LIN {X 0,Y 247.88,Z 687.786,A -85,B 0,C 180,E1 -19070.205,E2 -19070.205} C_VEL
LIN {X 0,Y 249.229,Z 685.586,A -85,B 0,C 180,E1 -19073.523,E2 -19073.523} C_VEL
LIN {X 0,Y 251.079,Z 682.164,A -85,B 0,C 180,E1 -19076.79,E2 -19076.79} C_VEL
LIN {X 0,Y 253.652,Z 677.44,A -85,B 0,C 180,E1 -19080,E2 -19080} C_VEL
LIN {X 0,Y 256.854,Z 671.391,A -85,B 0,C 180,E1 -19083.137,E2 -19083.137} C_VEL
LIN {X 0,Y 260.765,Z 663.772,A -85,B 0,C 180,E1 -19086.188,E2 -19086.188} C_VEL
LIN {X 0,Y 264.838,Z 655.76,A -85,B 0,C 180,E1 -19088.777,E2 -19088.777} C_VEL
LIN {X 0,Y 267.711,Z 649.729,A -85,B 0,C 180,E1 -19090.41,E2 -19090.41} C_VEL
LIN {X 0,Y 268.928,Z 646.197,A -85,B 0,C 180,E1 -19091.383,E2 -19091.383} C_VEL
LIN {X 0,Y 270.336,Z 634.797,A -85,B 0,C 180,E1 -19094.806,E2 -19094.806} C_VEL
LIN {X 0,Y 271.75,Z 630.731,A -85,B 0,C 180,E1 -19095.669,E2 -19095.669} C_VEL
LIN {X 0,Y 276.734,Z 619.024,A -85,B 0,C 180,E1 -19097.552,E2 -19097.552} C_VEL
LIN {X 0,Y 281.807,Z 605.606,A -85,B 0,C 180,E1 -19099.296,E2 -19099.296} C_VEL
LIN {X 0,Y 286.56,Z 591.439,A -85,B 0,C 180,E1 -19100.778,E2 -19100.778} C_VEL
LIN {X 0,Y 290.862,Z 576.419,A -85,B 0,C 180,E1 -19101.994,E2 -19101.994} C_VEL
LIN {X 0,Y 294.362,Z 561.567,A -85,B 0,C 180,E1 -19102.921,E2 -19102.921} C_VEL
LIN {X 0,Y 297.341,Z 545.848,A -85,B 0,C 180,E1 -19103.645,E2 -19103.645} C_VEL
LIN {X 0,Y 308.948,Z 468.897,A -85,B 0,C 180,E1 -19106.327,E2 -19106.327} C_VEL
LIN {X 0,Y 307.213,Z 464.58,A -85,B 0,C 180,E1 -19107.92,E2 -19107.92} C_VEL
LIN {X 0,Y 305.635,Z 461.133,A -85,B 0,C 180,E1 -19109.693,E2 -19109.693} C_VEL
LIN {X 0,Y 304.433,Z 458.679,A -85,B 0,C 180,E1 -19111.555,E2 -19111.555} C_VEL
LIN {X 0,Y 303.585,Z 457.434,A -85,B 0,C 180,E1 -19113.752,E2 -19113.752} C_VEL
LIN {X 0,Y 303.382,Z 457.554,A -85,B 0,C 180,E1 -19115.824,E2 -19115.824} C_VEL
LIN {X 0,Y 303.96,Z 459.719,A -85,B 0,C 180,E1 -19118.511,E2 -19118.511} C_VEL
LIN {X 0,Y 304.573,Z 461.273,A -85,B 0,C 180,E1 -19119.738,E2 -19119.738} C_VEL
LIN {X 0,Y 305.975,Z 465.574,A -85,B 0,C 180,E1 -19121.819,E2 -19121.819} C_VEL
LIN {X 0,Y 307.607,Z 470.737,A -85,B 0,C 180,E1 -19123.621,E2 -19123.621} C_VEL
LIN {X 0,Y 308.482,Z 473.787,A -85,B 0,C 180,E1 -19124.465,E2 -19124.465} C_VEL
LIN {X 0,Y 296.017,Z 556.561,A -85,B 0,C 180,E1 -19127.358,E2 -19127.358} C_VEL
LIN {X 0,Y 292.723,Z 572.399,A -85,B 0,C 180,E1 -19128.104,E2 -19128.104} C_VEL
LIN {X 0,Y 288.495,Z 588.462,A -85,B 0,C 180,E1 -19129.101,E2 -19129.101} C_VEL
LIN {X 0,Y 283.818,Z 603.365,A -85,B 0,C 180,E1 -19130.328,E2 -19130.328} C_VEL
LIN {X 0,Y 278.241,Z 618.997,A -85,B 0,C 180,E1 -19131.996,E2 -19131.996} C_VEL
LIN {X 0,Y 272.662,Z 632.821,A -85,B 0,C 180,E1 -19133.868,E2 -19133.868} C_VEL
LIN {X 0,Y 266.356,Z 647.07,A -85,B 0,C 180,E1 -19136.349,E2 -19136.349} C_VEL
LIN {X 0,Y 261.075,Z 658.229,A -85,B 0,C 180,E1 -19138.786,E2 -19138.786} C_VEL
LIN {X 0,Y 255.836,Z 668.683,A -85,B 0,C 180,E1 -19141.623,E2 -19141.623} C_VEL
LIN {X 0,Y 251.787,Z 676.761,A -85,B 0,C 180,E1 -19144.362,E2 -19144.362} C_VEL
LIN {X 0,Y 248.026,Z 684.215,A -85,B 0,C 180,E1 -19147.507,E2 -19147.507} C_VEL
LIN {X 0,Y 244.834,Z 690.278,A -85,B 0,C 180,E1 -19150.722,E2 -19150.722} C_VEL
LIN {X 0,Y 242.981,Z 693.924,A -85,B 0,C 180,E1 -19153.185,E2 -19153.185} C_VEL
LIN {X 0,Y 241.338,Z 697.72,A -85,B 0,C 180,E1 -19156.526,E2 -19156.526} C_VEL
LIN {X 0,Y 240.312,Z 700.321,A -85,B 0,C 180,E1 -19159.891,E2 -19159.891} C_VEL
LIN {X 0,Y 239.794,Z 701.759,A -85,B 0,C 180,E1 -19163.265,E2 -19163.265} C_VEL
LIN {X 0,Y 239.757,Z 701.968,A -85,B 0,C 180,E1 -19166.637,E2 -19166.637} C_VEL
LIN {X 0,Y 239.893,Z 701.614,A -85,B 0,C 180,E1 -19168.319,E2 -19168.319} C_VEL
LIN {X 0,Y 239.926,Z 699.962,A -85,B 0,C 180,E1 -19171.676,E2 -19171.676} C_VEL
LIN {X 0,Y 239.941,Z 696.811,A -85,B 0,C 180,E1 -19175.209,E2 -19175.209} C_VEL
LIN {X 0,Y 240.087,Z 692.603,A -85,B 0,C 180,E1 -19178.414,E2 -19178.414} C_VEL
LIN {X 0,Y 240.543,Z 686.661,A -85,B 0,C 180,E1 -19181.799,E2 -19181.799} C_VEL
LIN {X 0,Y 241.434,Z 680.097,A -85,B 0,C 180,E1 -19184.753,E2 -19184.753} C_VEL
LIN {X 0,Y 242.744,Z 672.341,A -85,B 0,C 180,E1 -19187.608,E2 -19187.608} C_VEL
LIN {X 0,Y 244.273,Z 663.893,A -85,B 0,C 180,E1 -19190.194,E2 -19190.194} C_VEL
LIN {X 0,Y 246.574,Z 652.437,A -85,B 0,C 180,E1 -19193.071,E2 -19193.071} C_VEL
LIN {X 0,Y 248.822,Z 640.832,A -85,B 0,C 180,E1 -19195.466,E2 -19195.466} C_VEL
LIN {X 0,Y 251.171,Z 628.98,A -85,B 0,C 180,E1 -19197.493,E2 -19197.493} C_VEL
LIN {X 0,Y 253.722,Z 615.002,A -85,B 0,C 180,E1 -19199.447,E2 -19199.447} C_VEL
LIN {X 0,Y 256.022,Z 601.49,A -85,B 0,C 180,E1 -19200.974,E2 -19200.974} C_VEL
LIN {X 0,Y 258.145,Z 586.74,A -85,B 0,C 180,E1 -19202.304,E2 -19202.304} C_VEL
LIN {X 0,Y 260.031,Z 571.411,A -85,B 0,C 180,E1 -19203.353,E2 -19203.353} C_VEL
LIN {X 0,Y 261.5,Z 555.708,A -85,B 0,C 180,E1 -19204.124,E2 -19204.124} C_VEL
LIN {X 0,Y 268.174,Z 451.601,A -85,B 0,C 180,E1 -19207.78,E2 -19207.78} C_VEL
LIN {X 0,Y 267.38,Z 447.714,A -85,B 0,C 180,E1 -19208.028,E2 -19208.028} C_VEL
LIN {X 0,Y 257.514,Z 422.783,A -85,B 0,C 180,E1 -19210.24,E2 -19210.24} C_VEL
LIN {X 0,Y 249.94,Z 405.473,A -85,B 0,C 180,E1 -19212.023,E2 -19212.023} C_VEL
LIN {X 0,Y 243.579,Z 391.38,A -85,B 0,C 180,E1 -19213.612,E2 -19213.612} C_VEL
LIN {X 0,Y 241.939,Z 384.975,A -85,B 0,C 180,E1 -19216.029,E2 -19216.029} C_VEL
LIN {X 0,Y 241.93,Z 384.979,A -85,B 0,C 180,E1 -19220.276,E2 -19220.276} C_VEL
LIN {X 0,Y 241.966,Z 384.972,A -85,B 0,C 180,E1 -19224.486,E2 -19224.486} C_VEL
LIN {X 0,Y 241.936,Z 384.975,A -85,B 0,C 180,E1 -19228.475,E2 -19228.475} C_VEL
LIN {X 0,Y 241.938,Z 384.972,A -85,B 0,C 180,E1 -19232.305,E2 -19232.305} C_VEL
LIN {X 0,Y 241.969,Z 384.968,A -85,B 0,C 180,E1 -19236.007,E2 -19236.007} C_VEL
LIN {X 0,Y 241.971,Z 384.968,A -85,B 0,C 180,E1 -19239.603,E2 -19239.603} C_VEL
LIN {X 0,Y 242.092,Z 384.951,A -85,B 0,C 180,E1 -19243.324,E2 -19243.324} C_VEL
LIN {X 0,Y 242.139,Z 384.938,A -85,B 0,C 180,E1 -19248.278,E2 -19248.278} C_VEL
LIN {X 0,Y 242.354,Z 384.914,A -85,B 0,C 180,E1 -19251.663,E2 -19251.663} C_VEL
LIN {X 0,Y 242.382,Z 384.915,A -85,B 0,C 180,E1 -19253.34,E2 -19253.34} C_VEL
LIN {X 0,Y 242.603,Z 384.89,A -85,B 0,C 180,E1 -19258.34,E2 -19258.34} C_VEL
LIN {X 0,Y 242.603,Z 384.891,A -85,B 0,C 180,E1 -19261.661,E2 -19261.661} C_VEL
LIN {X 0,Y 242.386,Z 384.916,A -85,B 0,C 180,E1 -19266.661,E2 -19266.661} C_VEL
LIN {X 0,Y 242.247,Z 384.931,A -85,B 0,C 180,E1 -19270.025,E2 -19270.025} C_VEL
LIN {X 0,Y 242.095,Z 384.951,A -85,B 0,C 180,E1 -19275.146,E2 -19275.146} C_VEL
LIN {X 0,Y 242.007,Z 384.96,A -85,B 0,C 180,E1 -19278.63,E2 -19278.63} C_VEL
LIN {X 0,Y 241.961,Z 384.97,A -85,B 0,C 180,E1 -19282.185,E2 -19282.185} C_VEL
LIN {X 0,Y 241.975,Z 384.963,A -85,B 0,C 180,E1 -19285.828,E2 -19285.828} C_VEL
LIN {X 0,Y 241.952,Z 384.971,A -85,B 0,C 180,E1 -19289.591,E2 -19289.591} C_VEL
LIN {X 0,Y 241.969,Z 384.965,A -85,B 0,C 180,E1 -19293.495,E2 -19293.495} C_VEL
LIN {X 0,Y 241.97,Z 384.968,A -85,B 0,C 180,E1 -19297.586,E2 -19297.586} C_VEL
LIN {X 0,Y 241.91,Z 384.97,A -85,B 0,C 180,E1 -19301.929,E2 -19301.929} C_VEL
LIN {X 0,Y 241.892,Z 384.977,A -85,B 0,C 180,E1 -19306.583,E2 -19306.583} C_VEL
LIN {X 0,Y 241.968,Z 384.964,A -85,B 0,C 180,E1 -19311.649,E2 -19311.649} C_VEL
LIN {X 0,Y 241.968,Z 384.968,A -85,B 0,C 180,E1 -19314.489,E2 -19314.489} C_VEL
LIN {X 0,Y 241.943,Z 384.965,A -85,B 0,C 180,E1 -19318.479,E2 -19318.479} C_VEL
LIN {X 0,Y 241.948,Z 384.971,A -85,B 0,C 180,E1 -19322.308,E2 -19322.308} C_VEL
LIN {X 0,Y 241.984,Z 384.965,A -85,B 0,C 180,E1 -19326.011,E2 -19326.011} C_VEL
LIN {X 0,Y 242.019,Z 384.965,A -85,B 0,C 180,E1 -19329.609,E2 -19329.609} C_VEL
LIN {X 0,Y 242.115,Z 384.941,A -85,B 0,C 180,E1 -19333.319,E2 -19333.319} C_VEL
LIN {X 0,Y 242.155,Z 384.936,A -85,B 0,C 180,E1 -19336.577,E2 -19336.577} C_VEL
LIN {X 0,Y 242.343,Z 384.921,A -85,B 0,C 180,E1 -19340.407,E2 -19340.407} C_VEL
LIN {X 0,Y 242.398,Z 384.911,A -85,B 0,C 180,E1 -19343.343,E2 -19343.343} C_VEL
LIN {X 0,Y 242.622,Z 384.888,A -85,B 0,C 180,E1 -19348.343,E2 -19348.343} C_VEL
LIN {X 0,Y 242.621,Z 384.883,A -85,B 0,C 180,E1 -19351.662,E2 -19351.662} C_VEL
LIN {X 0,Y 242.403,Z 384.916,A -85,B 0,C 180,E1 -19356.662,E2 -19356.662} C_VEL
LIN {X 0,Y 242.27,Z 384.93,A -85,B 0,C 180,E1 -19360.026,E2 -19360.026} C_VEL
LIN {X 0,Y 242.112,Z 384.948,A -85,B 0,C 180,E1 -19365.147,E2 -19365.147} C_VEL
LIN {X 0,Y 242.044,Z 384.956,A -85,B 0,C 180,E1 -19368.629,E2 -19368.629} C_VEL
LIN {X 0,Y 242.007,Z 384.962,A -85,B 0,C 180,E1 -19372.183,E2 -19372.183} C_VEL
LIN {X 0,Y 241.995,Z 384.966,A -85,B 0,C 180,E1 -19376.756,E2 -19376.756} C_VEL
LIN {X 0,Y 242.034,Z 384.961,A -85,B 0,C 180,E1 -19377.628,E2 -19377.628} C_VEL
LIN {X 0,Y 243.106,Z 387.957,A -85,B 0,C 180,E1 -19377.964,E2 -19377.964} C_VEL
LIN {X 0,Y 254.638,Z 409.921,A -85,B 0,C 180,E1 -19380.548,E2 -19380.548} C_VEL
LIN {X 0,Y 260.374,Z 422.165,A -85,B 0,C 180,E1 -19381.812,E2 -19381.812} C_VEL
LIN {X 0,Y 268.163,Z 441.082,A -85,B 0,C 180,E1 -19383.506,E2 -19383.506} C_VEL
LIN {X 0,Y 261.391,Z 544.984,A -85,B 0,C 180,E1 -19387.16,E2 -19387.16} C_VEL
LIN {X 0,Y 259.827,Z 560.878,A -85,B 0,C 180,E1 -19388.019,E2 -19388.019} C_VEL
LIN {X 0,Y 257.976,Z 576.825,A -85,B 0,C 180,E1 -19389.221,E2 -19389.221} C_VEL
LIN {X 0,Y 255.654,Z 592.523,A -85,B 0,C 180,E1 -19390.758,E2 -19390.758} C_VEL
LIN {X 0,Y 253.408,Z 605.906,A -85,B 0,C 180,E1 -19392.403,E2 -19392.403} C_VEL
LIN {X 0,Y 250.916,Z 619.48,A -85,B 0,C 180,E1 -19394.448,E2 -19394.448} C_VEL
LIN {X 0,Y 248.588,Z 631.789,A -85,B 0,C 180,E1 -19396.717,E2 -19396.717} C_VEL
LIN {X 0,Y 246.446,Z 642.171,A -85,B 0,C 180,E1 -19399.011,E2 -19399.011} C_VEL
LIN {X 0,Y 244.425,Z 652.702,A -85,B 0,C 180,E1 -19401.815,E2 -19401.815} C_VEL
LIN {X 0,Y 242.777,Z 661.39,A -85,B 0,C 180,E1 -19404.621,E2 -19404.621} C_VEL
LIN {X 0,Y 241.533,Z 668.857,A -85,B 0,C 180,E1 -19407.55,E2 -19407.55} C_VEL
LIN {X 0,Y 240.741,Z 674.529,A -85,B 0,C 180,E1 -19410.245,E2 -19410.245} C_VEL
LIN {X 0,Y 240.186,Z 679.262,A -85,B 0,C 180,E1 -19413.028,E2 -19413.028} C_VEL
LIN {X 0,Y 239.715,Z 682.915,A -85,B 0,C 180,E1 -19415.766,E2 -19415.766} C_VEL
LIN {X 0,Y 239.447,Z 686.389,A -85,B 0,C 180,E1 -19419.377,E2 -19419.377} C_VEL
LIN {X 0,Y 239.498,Z 688.397,A -85,B 0,C 180,E1 -19422.935,E2 -19422.935} C_VEL
LIN {X 0,Y 239.883,Z 689.056,A -85,B 0,C 180,E1 -19426.444,E2 -19426.444} C_VEL
LIN {X 0,Y 240.675,Z 688.451,A -85,B 0,C 180,E1 -19429.909,E2 -19429.909} C_VEL
LIN {X 0,Y 242.053,Z 686.612,A -85,B 0,C 180,E1 -19433.33,E2 -19433.33} C_VEL
LIN {X 0,Y 243.902,Z 683.528,A -85,B 0,C 180,E1 -19436.696,E2 -19436.696} C_VEL
LIN {X 0,Y 246.518,Z 679.203,A -85,B 0,C 180,E1 -19440,E2 -19440} C_VEL
LIN {X 0,Y 249.783,Z 673.54,A -85,B 0,C 180,E1 -19443.225,E2 -19443.225} C_VEL
LIN {X 0,Y 253.794,Z 666.466,A -85,B 0,C 180,E1 -19446.359,E2 -19446.359} C_VEL
LIN {X 0,Y 257.915,Z 658.897,A -85,B 0,C 180,E1 -19449.014,E2 -19449.014} C_VEL
LIN {X 0,Y 262.61,Z 649.918,A -85,B 0,C 180,E1 -19451.578,E2 -19451.578} C_VEL
LIN {X 0,Y 267.686,Z 639.572,A -85,B 0,C 180,E1 -19453.972,E2 -19453.972} C_VEL
LIN {X 0,Y 271.75,Z 630.731,A -85,B 0,C 180,E1 -19455.669,E2 -19455.669} C_VEL
LIN {X 0,Y 273.213,Z 626.626,A -85,B 0,C 180,E1 -19456.512,E2 -19456.512} C_VEL
LIN {X 0,Y 275.152,Z 614.753,A -85,B 0,C 180,E1 -19459.27,E2 -19459.27} C_VEL
LIN {X 0,Y 276.382,Z 610.304,A -85,B 0,C 180,E1 -19460.027,E2 -19460.027} C_VEL
LIN {X 0,Y 276.968,Z 608.722,A -85,B 0,C 180,E1 -19460.234,E2 -19460.234} C_VEL
LIN {X 0,Y 282.024,Z 594.812,A -85,B 0,C 180,E1 -19461.744,E2 -19461.744} C_VEL
LIN {X 0,Y 286.38,Z 581.125,A -85,B 0,C 180,E1 -19462.928,E2 -19462.928} C_VEL
LIN {X 0,Y 290.018,Z 567.604,A -85,B 0,C 180,E1 -19463.852,E2 -19463.852} C_VEL
LIN {X 0,Y 293.521,Z 551.339,A -85,B 0,C 180,E1 -19464.692,E2 -19464.692} C_VEL
LIN {X 0,Y 306.022,Z 473.195,A -85,B 0,C 180,E1 -19467.45,E2 -19467.45} C_VEL
LIN {X 0,Y 304.117,Z 468.309,A -85,B 0,C 180,E1 -19469.655,E2 -19469.655} C_VEL
LIN {X 0,Y 302.839,Z 465.531,A -85,B 0,C 180,E1 -19471.741,E2 -19471.741} C_VEL
LIN {X 0,Y 302.066,Z 464.347,A -85,B 0,C 180,E1 -19473.945,E2 -19473.945} C_VEL
LIN {X 0,Y 301.907,Z 464.592,A -85,B 0,C 180,E1 -19475.977,E2 -19475.977} C_VEL
LIN {X 0,Y 302.48,Z 466.851,A -85,B 0,C 180,E1 -19478.591,E2 -19478.591} C_VEL
LIN {X 0,Y 302.861,Z 468.094,A -85,B 0,C 180,E1 -19479.481,E2 -19479.481} C_VEL
LIN {X 0,Y 303.977,Z 471.983,A -85,B 0,C 180,E1 -19481.373,E2 -19481.373} C_VEL
LIN {X 0,Y 305.294,Z 476.638,A -85,B 0,C 180,E1 -19483.026,E2 -19483.026} C_VEL
LIN {X 0,Y 305.571,Z 477.721,A -85,B 0,C 180,E1 -19483.342,E2 -19483.342} C_VEL
LIN {X 0,Y 293.012,Z 556.809,A -85,B 0,C 180,E1 -19486.104,E2 -19486.104} C_VEL
LIN {X 0,Y 289.914,Z 571.167,A -85,B 0,C 180,E1 -19486.776,E2 -19486.776} C_VEL
LIN {X 0,Y 285.639,Z 586.713,A -85,B 0,C 180,E1 -19487.716,E2 -19487.716} C_VEL
LIN {X 0,Y 280.729,Z 601.757,A -85,B 0,C 180,E1 -19488.914,E2 -19488.914} C_VEL
LIN {X 0,Y 275.464,Z 615.934,A -85,B 0,C 180,E1 -19490.367,E2 -19490.367} C_VEL
LIN {X 0,Y 269.538,Z 630.011,A -85,B 0,C 180,E1 -19492.21,E2 -19492.21} C_VEL
LIN {X 0,Y 264.115,Z 641.993,A -85,B 0,C 180,E1 -19494.166,E2 -19494.166} C_VEL
LIN {X 0,Y 259.08,Z 652.225,A -85,B 0,C 180,E1 -19496.211,E2 -19496.211} C_VEL
LIN {X 0,Y 253.7,Z 662.524,A -85,B 0,C 180,E1 -19498.705,E2 -19498.705} C_VEL
LIN {X 0,Y 248.935,Z 671.26,A -85,B 0,C 180,E1 -19501.316,E2 -19501.316} C_VEL
LIN {X 0,Y 244.378,Z 679.622,A -85,B 0,C 180,E1 -19504.442,E2 -19504.442} C_VEL
LIN {X 0,Y 240.604,Z 686.476,A -85,B 0,C 180,E1 -19507.681,E2 -19507.681} C_VEL
LIN {X 0,Y 237.393,Z 692.002,A -85,B 0,C 180,E1 -19510.992,E2 -19510.992} C_VEL
LIN {X 0,Y 235.258,Z 696.205,A -85,B 0,C 180,E1 -19514.401,E2 -19514.401} C_VEL
LIN {X 0,Y 233.715,Z 699.218,A -85,B 0,C 180,E1 -19517.846,E2 -19517.846} C_VEL
LIN {X 0,Y 232.949,Z 701.078,A -85,B 0,C 180,E1 -19521.321,E2 -19521.321} C_VEL
LIN {X 0,Y 232.646,Z 701.784,A -85,B 0,C 180,E1 -19524.798,E2 -19524.798} C_VEL
LIN {X 0,Y 232.798,Z 701.286,A -85,B 0,C 180,E1 -19528.267,E2 -19528.267} C_VEL
LIN {X 0,Y 232.848,Z 700.548,A -85,B 0,C 180,E1 -19529.997,E2 -19529.997} C_VEL
LIN {X 0,Y 232.858,Z 699.488,A -85,B 0,C 180,E1 -19531.727,E2 -19531.727} C_VEL
LIN {X 0,Y 232.878,Z 696.368,A -85,B 0,C 180,E1 -19535.192,E2 -19535.192} C_VEL
LIN {X 0,Y 233.02,Z 691.824,A -85,B 0,C 180,E1 -19538.671,E2 -19538.671} C_VEL
LIN {X 0,Y 233.545,Z 685.73,A -85,B 0,C 180,E1 -19542.158,E2 -19542.158} C_VEL
LIN {X 0,Y 234.483,Z 678.999,A -85,B 0,C 180,E1 -19545.201,E2 -19545.201} C_VEL
LIN {X 0,Y 235.945,Z 670.799,A -85,B 0,C 180,E1 -19548.223,E2 -19548.223} C_VEL
LIN {X 0,Y 237.867,Z 660.853,A -85,B 0,C 180,E1 -19551.216,E2 -19551.216} C_VEL
LIN {X 0,Y 239.931,Z 650.663,A -85,B 0,C 180,E1 -19553.748,E2 -19553.748} C_VEL
LIN {X 0,Y 242.137,Z 639.638,A -85,B 0,C 180,E1 -19556.037,E2 -19556.037} C_VEL
LIN {X 0,Y 244.514,Z 627.848,A -85,B 0,C 180,E1 -19558.074,E2 -19558.074} C_VEL
LIN {X 0,Y 246.881,Z 615.258,A -85,B 0,C 180,E1 -19559.876,E2 -19559.876} C_VEL
LIN {X 0,Y 249.229,Z 601.848,A -85,B 0,C 180,E1 -19561.442,E2 -19561.442} C_VEL
LIN {X 0,Y 251.34,Z 587.946,A -85,B 0,C 180,E1 -19562.746,E2 -19562.746} C_VEL
LIN {X 0,Y 253.369,Z 572.224,A -85,B 0,C 180,E1 -19563.87,E2 -19563.87} C_VEL
LIN {X 0,Y 254.826,Z 556.973,A -85,B 0,C 180,E1 -19564.665,E2 -19564.665} C_VEL
LIN {X 0,Y 261.743,Z 452.264,A -85,B 0,C 180,E1 -19568.45,E2 -19568.45} C_VEL
LIN {X 0,Y 259.763,Z 446.226,A -85,B 0,C 180,E1 -19568.937,E2 -19568.937} C_VEL
LIN {X 0,Y 249.571,Z 420.785,A -85,B 0,C 180,E1 -19571.354,E2 -19571.354} C_VEL
LIN {X 0,Y 239.424,Z 398.251,A -85,B 0,C 180,E1 -19573.825,E2 -19573.825} C_VEL
LIN {X 0,Y 236.247,Z 391.245,A -85,B 0,C 180,E1 -19574.684,E2 -19574.684} C_VEL
LIN {X 0,Y 234.906,Z 385.85,A -85,B 0,C 180,E1 -19576.78,E2 -19576.78} C_VEL
LIN {X 0,Y 234.907,Z 385.851,A -85,B 0,C 180,E1 -19581.077,E2 -19581.077} C_VEL
LIN {X 0,Y 234.913,Z 385.849,A -85,B 0,C 180,E1 -19585.36,E2 -19585.36} C_VEL
LIN {X 0,Y 234.882,Z 385.852,A -85,B 0,C 180,E1 -19589.426,E2 -19589.426} C_VEL
LIN {X 0,Y 234.927,Z 385.841,A -85,B 0,C 180,E1 -19593.82,E2 -19593.82} C_VEL
LIN {X 0,Y 234.923,Z 385.845,A -85,B 0,C 180,E1 -19598.962,E2 -19598.962} C_VEL
LIN {X 0,Y 235.036,Z 385.829,A -85,B 0,C 180,E1 -19603.097,E2 -19603.097} C_VEL
LIN {X 0,Y 235.071,Z 385.821,A -85,B 0,C 180,E1 -19607.92,E2 -19607.92} C_VEL
LIN {X 0,Y 235.291,Z 385.793,A -85,B 0,C 180,E1 -19611.411,E2 -19611.411} C_VEL
LIN {X 0,Y 235.333,Z 385.793,A -85,B 0,C 180,E1 -19613.14,E2 -19613.14} C_VEL
LIN {X 0,Y 235.562,Z 385.767,A -85,B 0,C 180,E1 -19618.291,E2 -19618.291} C_VEL
LIN {X 0,Y 235.562,Z 385.768,A -85,B 0,C 180,E1 -19621.71,E2 -19621.71} C_VEL
LIN {X 0,Y 235.338,Z 385.794,A -85,B 0,C 180,E1 -19626.861,E2 -19626.861} C_VEL
LIN {X 0,Y 235.171,Z 385.811,A -85,B 0,C 180,E1 -19630.33,E2 -19630.33} C_VEL
LIN {X 0,Y 235.047,Z 385.831,A -85,B 0,C 180,E1 -19635.611,E2 -19635.611} C_VEL
LIN {X 0,Y 234.948,Z 385.839,A -85,B 0,C 180,E1 -19639.211,E2 -19639.211} C_VEL
LIN {X 0,Y 234.905,Z 385.846,A -85,B 0,C 180,E1 -19642.889,E2 -19642.889} C_VEL
LIN {X 0,Y 234.911,Z 385.842,A -85,B 0,C 180,E1 -19646.665,E2 -19646.665} C_VEL
LIN {X 0,Y 234.884,Z 385.85,A -85,B 0,C 180,E1 -19650.575,E2 -19650.575} C_VEL
LIN {X 0,Y 234.915,Z 385.84,A -85,B 0,C 180,E1 -19654.641,E2 -19654.641} C_VEL
LIN {X 0,Y 234.903,Z 385.847,A -85,B 0,C 180,E1 -19658.937,E2 -19658.937} C_VEL
LIN {X 0,Y 234.853,Z 385.848,A -85,B 0,C 180,E1 -19663.495,E2 -19663.495} C_VEL
LIN {X 0,Y 234.845,Z 385.855,A -85,B 0,C 180,E1 -19666.508,E2 -19666.508} C_VEL
LIN {X 0,Y 234.912,Z 385.839,A -85,B 0,C 180,E1 -19671.081,E2 -19671.081} C_VEL
LIN {X 0,Y 234.917,Z 385.847,A -85,B 0,C 180,E1 -19675.363,E2 -19675.363} C_VEL
LIN {X 0,Y 234.89,Z 385.845,A -85,B 0,C 180,E1 -19679.43,E2 -19679.43} C_VEL
LIN {X 0,Y 234.937,Z 385.844,A -85,B 0,C 180,E1 -19683.824,E2 -19683.824} C_VEL
LIN {X 0,Y 234.966,Z 385.841,A -85,B 0,C 180,E1 -19688.969,E2 -19688.969} C_VEL
LIN {X 0,Y 235.056,Z 385.822,A -85,B 0,C 180,E1 -19693.095,E2 -19693.095} C_VEL
LIN {X 0,Y 235.111,Z 385.82,A -85,B 0,C 180,E1 -19697.925,E2 -19697.925} C_VEL
LIN {X 0,Y 235.313,Z 385.799,A -85,B 0,C 180,E1 -19701.414,E2 -19701.414} C_VEL
LIN {X 0,Y 235.349,Z 385.79,A -85,B 0,C 180,E1 -19703.142,E2 -19703.142} C_VEL
LIN {X 0,Y 235.581,Z 385.765,A -85,B 0,C 180,E1 -19708.293,E2 -19708.293} C_VEL
LIN {X 0,Y 235.58,Z 385.759,A -85,B 0,C 180,E1 -19711.712,E2 -19711.712} C_VEL
LIN {X 0,Y 235.354,Z 385.795,A -85,B 0,C 180,E1 -19716.863,E2 -19716.863} C_VEL
LIN {X 0,Y 235.216,Z 385.809,A -85,B 0,C 180,E1 -19720.33,E2 -19720.33} C_VEL
LIN {X 0,Y 235.064,Z 385.829,A -85,B 0,C 180,E1 -19725.612,E2 -19725.612} C_VEL
LIN {X 0,Y 234.987,Z 385.836,A -85,B 0,C 180,E1 -19729.21,E2 -19729.21} C_VEL
LIN {X 0,Y 234.946,Z 385.843,A -85,B 0,C 180,E1 -19732.887,E2 -19732.887} C_VEL
LIN {X 0,Y 234.947,Z 385.844,A -85,B 0,C 180,E1 -19736.622,E2 -19736.622} C_VEL
LIN {X 0,Y 236.012,Z 388.749,A -85,B 0,C 180,E1 -19736.951,E2 -19736.951} C_VEL
LIN {X 0,Y 245.134,Z 405.869,A -85,B 0,C 180,E1 -19739.113,E2 -19739.113} C_VEL
LIN {X 0,Y 254.074,Z 424.079,A -85,B 0,C 180,E1 -19741.121,E2 -19741.121} C_VEL
LIN {X 0,Y 261.689,Z 442.792,A -85,B 0,C 180,E1 -19742.858,E2 -19742.858} C_VEL
LIN {X 0,Y 254.839,Z 545.121,A -85,B 0,C 180,E1 -19746.561,E2 -19746.561} C_VEL
LIN {X 0,Y 253.405,Z 559.639,A -85,B 0,C 180,E1 -19747.348,E2 -19747.348} C_VEL
LIN {X 0,Y 251.53,Z 575.326,A -85,B 0,C 180,E1 -19748.523,E2 -19748.523} C_VEL
LIN {X 0,Y 249.326,Z 590.237,A -85,B 0,C 180,E1 -19749.971,E2 -19749.971} C_VEL
LIN {X 0,Y 246.957,Z 604.162,A -85,B 0,C 180,E1 -19751.665,E2 -19751.665} C_VEL
LIN {X 0,Y 244.422,Z 617.892,A -85,B 0,C 180,E1 -19753.732,E2 -19753.732} C_VEL
LIN {X 0,Y 241.913,Z 630.767,A -85,B 0,C 180,E1 -19756.11,E2 -19756.11} C_VEL
LIN {X 0,Y 239.506,Z 642.24,A -85,B 0,C 180,E1 -19758.682,E2 -19758.682} C_VEL
LIN {X 0,Y 237.407,Z 652.772,A -85,B 0,C 180,E1 -19761.561,E2 -19761.561} C_VEL
LIN {X 0,Y 235.738,Z 661.481,A -85,B 0,C 180,E1 -19764.454,E2 -19764.454} C_VEL
LIN {X 0,Y 234.342,Z 669.777,A -85,B 0,C 180,E1 -19767.836,E2 -19767.836} C_VEL
LIN {X 0,Y 233.419,Z 676.327,A -85,B 0,C 180,E1 -19771.2,E2 -19771.2} C_VEL
LIN {X 0,Y 232.888,Z 680.716,A -85,B 0,C 180,E1 -19774.051,E2 -19774.051} C_VEL
LIN {X 0,Y 232.454,Z 684.107,A -85,B 0,C 180,E1 -19776.856,E2 -19776.856} C_VEL
LIN {X 0,Y 232.326,Z 687.238,A -85,B 0,C 180,E1 -19780.563,E2 -19780.563} C_VEL
LIN {X 0,Y 232.501,Z 688.912,A -85,B 0,C 180,E1 -19784.213,E2 -19784.213} C_VEL
LIN {X 0,Y 233.018,Z 689.267,A -85,B 0,C 180,E1 -19787.811,E2 -19787.811} C_VEL
LIN {X 0,Y 234.303,Z 688.173,A -85,B 0,C 180,E1 -19791.841,E2 -19791.841} C_VEL
LIN {X 0,Y 235.672,Z 686.289,A -85,B 0,C 180,E1 -19794.867,E2 -19794.867} C_VEL
LIN {X 0,Y 237.956,Z 682.995,A -85,B 0,C 180,E1 -19798.307,E2 -19798.307} C_VEL
LIN {X 0,Y 240.926,Z 678.434,A -85,B 0,C 180,E1 -19801.671,E2 -19801.671} C_VEL
LIN {X 0,Y 244.642,Z 672.569,A -85,B 0,C 180,E1 -19804.944,E2 -19804.944} C_VEL
LIN {X 0,Y 249.142,Z 665.161,A -85,B 0,C 180,E1 -19808.108,E2 -19808.108} C_VEL
LIN {X 0,Y 253.725,Z 657.352,A -85,B 0,C 180,E1 -19810.776,E2 -19810.776} C_VEL
LIN {X 0,Y 258.818,Z 648.03,A -85,B 0,C 180,E1 -19813.344,E2 -19813.344} C_VEL
LIN {X 0,Y 264.514,Z 637.022,A -85,B 0,C 180,E1 -19815.803,E2 -19815.803} C_VEL
LIN {X 0,Y 270.253,Z 624.759,A -85,B 0,C 180,E1 -19817.987,E2 -19817.987} C_VEL
LIN {X 0,Y 275.602,Z 612.271,A -85,B 0,C 180,E1 -19819.786,E2 -19819.786} C_VEL
LIN {X 0,Y 276.968,Z 608.722,A -85,B 0,C 180,E1 -19820.234,E2 -19820.234} C_VEL
LIN {X 0,Y 277.872,Z 605.639,A -85,B 0,C 180,E1 -19820.725,E2 -19820.725} C_VEL
LIN {X 0,Y 278.565,Z 596.621,A -85,B 0,C 180,E1 -19822.794,E2 -19822.794} C_VEL
LIN {X 0,Y 279.424,Z 593.394,A -85,B 0,C 180,E1 -19823.237,E2 -19823.237} C_VEL
LIN {X 0,Y 284.267,Z 578.423,A -85,B 0,C 180,E1 -19824.463,E2 -19824.463} C_VEL
LIN {X 0,Y 288.074,Z 564.569,A -85,B 0,C 180,E1 -19825.353,E2 -19825.353} C_VEL
LIN {X 0,Y 291.605,Z 548.16,A -85,B 0,C 180,E1 -19826.133,E2 -19826.133} C_VEL
LIN {X 0,Y 303.352,Z 478.07,A -85,B 0,C 180,E1 -19828.57,E2 -19828.57} C_VEL
LIN {X 0,Y 302.289,Z 474.84,A -85,B 0,C 180,E1 -19830.055,E2 -19830.055} C_VEL
LIN {X 0,Y 301.249,Z 472.363,A -85,B 0,C 180,E1 -19831.928,E2 -19831.928} C_VEL
LIN {X 0,Y 300.682,Z 471.449,A -85,B 0,C 180,E1 -19833.356,E2 -19833.356} C_VEL
LIN {X 0,Y 300.404,Z 471.447,A -85,B 0,C 180,E1 -19835.794,E2 -19835.794} C_VEL
LIN {X 0,Y 300.889,Z 473.712,A -85,B 0,C 180,E1 -19838.407,E2 -19838.407} C_VEL
LIN {X 0,Y 301.298,Z 475.468,A -85,B 0,C 180,E1 -19839.516,E2 -19839.516} C_VEL
LIN {X 0,Y 302.161,Z 478.839,A -85,B 0,C 180,E1 -19841.105,E2 -19841.105} C_VEL
LIN {X 0,Y 302.933,Z 481.857,A -85,B 0,C 180,E1 -19842.18,E2 -19842.18} C_VEL
LIN {X 0,Y 290.514,Z 556.084,A -85,B 0,C 180,E1 -19844.773,E2 -19844.773} C_VEL
LIN {X 0,Y 287.297,Z 570.283,A -85,B 0,C 180,E1 -19845.429,E2 -19845.429} C_VEL
LIN {X 0,Y 283.012,Z 585.339,A -85,B 0,C 180,E1 -19846.315,E2 -19846.315} C_VEL
LIN {X 0,Y 277.871,Z 600.527,A -85,B 0,C 180,E1 -19847.48,E2 -19847.48} C_VEL
LIN {X 0,Y 272.49,Z 614.341,A -85,B 0,C 180,E1 -19848.874,E2 -19848.874} C_VEL
LIN {X 0,Y 266.239,Z 628.608,A -85,B 0,C 180,E1 -19850.686,E2 -19850.686} C_VEL
LIN {X 0,Y 261.391,Z 638.78,A -85,B 0,C 180,E1 -19852.287,E2 -19852.287} C_VEL
LIN {X 0,Y 255.076,Z 650.971,A -85,B 0,C 180,E1 -19854.645,E2 -19854.645} C_VEL
LIN {X 0,Y 249.316,Z 661.336,A -85,B 0,C 180,E1 -19857.134,E2 -19857.134} C_VEL
LIN {X 0,Y 243.775,Z 670.822,A -85,B 0,C 180,E1 -19859.976,E2 -19859.976} C_VEL
LIN {X 0,Y 239.161,Z 678.628,A -85,B 0,C 180,E1 -19862.901,E2 -19862.901} C_VEL
LIN {X 0,Y 235.007,Z 685.573,A -85,B 0,C 180,E1 -19866.186,E2 -19866.186} C_VEL
LIN {X 0,Y 231.458,Z 691.171,A -85,B 0,C 180,E1 -19869.56,E2 -19869.56} C_VEL
LIN {X 0,Y 229.35,Z 694.553,A -85,B 0,C 180,E1 -19872.153,E2 -19872.153} C_VEL
LIN {X 0,Y 227.494,Z 698.022,A -85,B 0,C 180,E1 -19875.689,E2 -19875.689} C_VEL
LIN {X 0,Y 226.228,Z 700.271,A -85,B 0,C 180,E1 -19879.255,E2 -19879.255} C_VEL
LIN {X 0,Y 225.652,Z 701.393,A -85,B 0,C 180,E1 -19882.841,E2 -19882.841} C_VEL
LIN {X 0,Y 225.59,Z 701.356,A -85,B 0,C 180,E1 -19886.425,E2 -19886.425} C_VEL
LIN {X 0,Y 225.706,Z 700.893,A -85,B 0,C 180,E1 -19888.213,E2 -19888.213} C_VEL
LIN {X 0,Y 225.781,Z 700.119,A -85,B 0,C 180,E1 -19889.997,E2 -19889.997} C_VEL
LIN {X 0,Y 225.791,Z 699.008,A -85,B 0,C 180,E1 -19891.781,E2 -19891.781} C_VEL
LIN {X 0,Y 225.795,Z 695.735,A -85,B 0,C 180,E1 -19895.355,E2 -19895.355} C_VEL
LIN {X 0,Y 225.951,Z 691.018,A -85,B 0,C 180,E1 -19898.944,E2 -19898.944} C_VEL
LIN {X 0,Y 226.548,Z 684.741,A -85,B 0,C 180,E1 -19902.539,E2 -19902.539} C_VEL
LIN {X 0,Y 227.554,Z 677.81,A -85,B 0,C 180,E1 -19905.676,E2 -19905.676} C_VEL
LIN {X 0,Y 229.124,Z 669.405,A -85,B 0,C 180,E1 -19908.785,E2 -19908.785} C_VEL
LIN {X 0,Y 231.132,Z 659.229,A -85,B 0,C 180,E1 -19911.866,E2 -19911.866} C_VEL
LIN {X 0,Y 233.294,Z 648.781,A -85,B 0,C 180,E1 -19914.467,E2 -19914.467} C_VEL
LIN {X 0,Y 235.698,Z 637.487,A -85,B 0,C 180,E1 -19916.804,E2 -19916.804} C_VEL
LIN {X 0,Y 238.43,Z 624.031,A -85,B 0,C 180,E1 -19919.098,E2 -19919.098} C_VEL
LIN {X 0,Y 240.935,Z 610.748,A -85,B 0,C 180,E1 -19920.935,E2 -19920.935} C_VEL
LIN {X 0,Y 243.587,Z 595.469,A -85,B 0,C 180,E1 -19922.624,E2 -19922.624} C_VEL
LIN {X 0,Y 245.798,Z 579.823,A -85,B 0,C 180,E1 -19923.954,E2 -19923.954} C_VEL
LIN {X 0,Y 247.654,Z 563.903,A -85,B 0,C 180,E1 -19924.948,E2 -19924.948} C_VEL
LIN {X 0,Y 249.069,Z 546.189,A -85,B 0,C 180,E1 -19925.711,E2 -19925.711} C_VEL
LIN {X 0,Y 255.379,Z 453.331,A -85,B 0,C 180,E1 -19929.134,E2 -19929.134} C_VEL
LIN {X 0,Y 246.046,Z 429.434,A -85,B 0,C 180,E1 -19931.394,E2 -19931.394} C_VEL
LIN {X 0,Y 236.311,Z 406.954,A -85,B 0,C 180,E1 -19933.839,E2 -19933.839} C_VEL
LIN {X 0,Y 228.915,Z 390.974,A -85,B 0,C 180,E1 -19935.851,E2 -19935.851} C_VEL
LIN {X 0,Y 227.816,Z 386.734,A -85,B 0,C 180,E1 -19937.583,E2 -19937.583} C_VEL
LIN {X 0,Y 227.828,Z 386.735,A -85,B 0,C 180,E1 -19941.906,E2 -19941.906} C_VEL
LIN {X 0,Y 227.867,Z 386.729,A -85,B 0,C 180,E1 -19946.376,E2 -19946.376} C_VEL
LIN {X 0,Y 227.859,Z 386.727,A -85,B 0,C 180,E1 -19950.43,E2 -19950.43} C_VEL
LIN {X 0,Y 227.858,Z 386.72,A -85,B 0,C 180,E1 -19954.418,E2 -19954.418} C_VEL
LIN {X 0,Y 227.906,Z 386.722,A -85,B 0,C 180,E1 -19958.282,E2 -19958.282} C_VEL
LIN {X 0,Y 227.996,Z 386.709,A -85,B 0,C 180,E1 -19963.894,E2 -19963.894} C_VEL
LIN {X 0,Y 228.112,Z 386.681,A -85,B 0,C 180,E1 -19969.348,E2 -19969.348} C_VEL
LIN {X 0,Y 228.285,Z 386.671,A -85,B 0,C 180,E1 -19972.927,E2 -19972.927} C_VEL
LIN {X 0,Y 228.52,Z 386.644,A -85,B 0,C 180,E1 -19978.238,E2 -19978.238} C_VEL
LIN {X 0,Y 228.52,Z 386.645,A -85,B 0,C 180,E1 -19981.763,E2 -19981.763} C_VEL
LIN {X 0,Y 228.291,Z 386.672,A -85,B 0,C 180,E1 -19987.074,E2 -19987.074} C_VEL
LIN {X 0,Y 228.112,Z 386.69,A -85,B 0,C 180,E1 -19990.653,E2 -19990.653} C_VEL
LIN {X 0,Y 227.997,Z 386.706,A -85,B 0,C 180,E1 -19996.107,E2 -19996.107} C_VEL
LIN {X 0,Y 227.908,Z 386.722,A -85,B 0,C 180,E1 -20001.719,E2 -20001.719} C_VEL
LIN {X 0,Y 227.89,Z 386.717,A -85,B 0,C 180,E1 -20006.583,E2 -20006.583} C_VEL
LIN {X 0,Y 227.859,Z 386.726,A -85,B 0,C 180,E1 -20010.281,E2 -20010.281} C_VEL
LIN {X 0,Y 227.867,Z 386.719,A -85,B 0,C 180,E1 -20013.723,E2 -20013.723} C_VEL
LIN {X 0,Y 227.831,Z 386.73,A -85,B 0,C 180,E1 -20018.094,E2 -20018.094} C_VEL
LIN {X 0,Y 227.784,Z 386.726,A -85,B 0,C 180,E1 -20022.749,E2 -20022.749} C_VEL
LIN {X 0,Y 227.776,Z 386.736,A -85,B 0,C 180,E1 -20027.254,E2 -20027.254} C_VEL
LIN {X 0,Y 227.831,Z 386.726,A -85,B 0,C 180,E1 -20031.91,E2 -20031.91} C_VEL
LIN {X 0,Y 227.873,Z 386.722,A -85,B 0,C 180,E1 -20036.381,E2 -20036.381} C_VEL
LIN {X 0,Y 227.867,Z 386.724,A -85,B 0,C 180,E1 -20040.434,E2 -20040.434} C_VEL
LIN {X 0,Y 227.869,Z 386.721,A -85,B 0,C 180,E1 -20044.422,E2 -20044.422} C_VEL
LIN {X 0,Y 227.94,Z 386.717,A -85,B 0,C 180,E1 -20048.288,E2 -20048.288} C_VEL
LIN {X 0,Y 228.024,Z 386.687,A -85,B 0,C 180,E1 -20053.898,E2 -20053.898} C_VEL
LIN {X 0,Y 228.068,Z 386.693,A -85,B 0,C 180,E1 -20057.546,E2 -20057.546} C_VEL
LIN {X 0,Y 228.254,Z 386.677,A -85,B 0,C 180,E1 -20061.147,E2 -20061.147} C_VEL
LIN {X 0,Y 228.302,Z 386.667,A -85,B 0,C 180,E1 -20062.93,E2 -20062.93} C_VEL
LIN {X 0,Y 228.539,Z 386.643,A -85,B 0,C 180,E1 -20068.24,E2 -20068.24} C_VEL
LIN {X 0,Y 228.538,Z 386.636,A -85,B 0,C 180,E1 -20071.765,E2 -20071.765} C_VEL
LIN {X 0,Y 228.307,Z 386.673,A -85,B 0,C 180,E1 -20077.075,E2 -20077.075} C_VEL
LIN {X 0,Y 228.145,Z 386.689,A -85,B 0,C 180,E1 -20080.654,E2 -20080.654} C_VEL
LIN {X 0,Y 228.015,Z 386.708,A -85,B 0,C 180,E1 -20086.108,E2 -20086.108} C_VEL
LIN {X 0,Y 227.956,Z 386.712,A -85,B 0,C 180,E1 -20091.716,E2 -20091.716} C_VEL
LIN {X 0,Y 227.887,Z 386.721,A -85,B 0,C 180,E1 -20095.582,E2 -20095.582} C_VEL
LIN {X 0,Y 228.967,Z 389.691,A -85,B 0,C 180,E1 -20095.919,E2 -20095.919} C_VEL
LIN {X 0,Y 236.787,Z 404.157,A -85,B 0,C 180,E1 -20097.849,E2 -20097.849} C_VEL
LIN {X 0,Y 247.403,Z 425.27,A -85,B 0,C 180,E1 -20100.333,E2 -20100.333} C_VEL
LIN {X 0,Y 255.318,Z 444.708,A -85,B 0,C 180,E1 -20102.202,E2 -20102.202} C_VEL
LIN {X 0,Y 248.307,Z 545.265,A -85,B 0,C 180,E1 -20105.93,E2 -20105.93} C_VEL
LIN {X 0,Y 246.656,Z 561.176,A -85,B 0,C 180,E1 -20106.838,E2 -20106.838} C_VEL
LIN {X 0,Y 244.802,Z 576.313,A -85,B 0,C 180,E1 -20108.028,E2 -20108.028} C_VEL
LIN {X 0,Y 242.58,Z 590.75,A -85,B 0,C 180,E1 -20109.479,E2 -20109.479} C_VEL
LIN {X 0,Y 239.969,Z 605.635,A -85,B 0,C 180,E1 -20111.367,E2 -20111.367} C_VEL
LIN {X 0,Y 237.328,Z 619.128,A -85,B 0,C 180,E1 -20113.487,E2 -20113.487} C_VEL
LIN {X 0,Y 234.827,Z 631.721,A -85,B 0,C 180,E1 -20115.916,E2 -20115.916} C_VEL
LIN {X 0,Y 232.352,Z 643.214,A -85,B 0,C 180,E1 -20118.603,E2 -20118.603} C_VEL
LIN {X 0,Y 230.418,Z 652.74,A -85,B 0,C 180,E1 -20121.297,E2 -20121.297} C_VEL
LIN {X 0,Y 228.677,Z 661.491,A -85,B 0,C 180,E1 -20124.272,E2 -20124.272} C_VEL
LIN {X 0,Y 227.384,Z 668.957,A -85,B 0,C 180,E1 -20127.352,E2 -20127.352} C_VEL
LIN {X 0,Y 226.517,Z 674.875,A -85,B 0,C 180,E1 -20130.317,E2 -20130.317} C_VEL
LIN {X 0,Y 225.963,Z 679.509,A -85,B 0,C 180,E1 -20133.192,E2 -20133.192} C_VEL
LIN {X 0,Y 225.465,Z 683.22,A -85,B 0,C 180,E1 -20136.094,E2 -20136.094} C_VEL
LIN {X 0,Y 225.267,Z 686.742,A -85,B 0,C 180,E1 -20139.928,E2 -20139.928} C_VEL
LIN {X 0,Y 225.348,Z 688.808,A -85,B 0,C 180,E1 -20143.698,E2 -20143.698} C_VEL
LIN {X 0,Y 225.858,Z 689.553,A -85,B 0,C 180,E1 -20147.419,E2 -20147.419} C_VEL
LIN {X 0,Y 226.884,Z 689.044,A -85,B 0,C 180,E1 -20151.09,E2 -20151.09} C_VEL
LIN {X 0,Y 228.465,Z 687.305,A -85,B 0,C 180,E1 -20154.704,E2 -20154.704} C_VEL
LIN {X 0,Y 230.753,Z 684.351,A -85,B 0,C 180,E1 -20158.254,E2 -20158.254} C_VEL
LIN {X 0,Y 233.788,Z 680.208,A -85,B 0,C 180,E1 -20161.722,E2 -20161.722} C_VEL
LIN {X 0,Y 237.569,Z 674.745,A -85,B 0,C 180,E1 -20165.091,E2 -20165.091} C_VEL
LIN {X 0,Y 242.155,Z 667.904,A -85,B 0,C 180,E1 -20168.343,E2 -20168.343} C_VEL
LIN {X 0,Y 246.86,Z 660.573,A -85,B 0,C 180,E1 -20171.079,E2 -20171.079} C_VEL
LIN {X 0,Y 252.082,Z 651.932,A -85,B 0,C 180,E1 -20173.708,E2 -20173.708} C_VEL
LIN {X 0,Y 257.933,Z 641.573,A -85,B 0,C 180,E1 -20176.217,E2 -20176.217} C_VEL
LIN {X 0,Y 264.294,Z 629.262,A -85,B 0,C 180,E1 -20178.608,E2 -20178.608} C_VEL
LIN {X 0,Y 269.857,Z 617.35,A -85,B 0,C 180,E1 -20180.46,E2 -20180.46} C_VEL
LIN {X 0,Y 275.642,Z 603.53,A -85,B 0,C 180,E1 -20182.191,E2 -20182.191} C_VEL
LIN {X 0,Y 279.424,Z 593.394,A -85,B 0,C 180,E1 -20183.237,E2 -20183.237} C_VEL
LIN {X 0,Y 280.913,Z 588.416,A -85,B 0,C 180,E1 -20183.815,E2 -20183.815} C_VEL
LIN {X 0,Y 283.61,Z 573.276,A -85,B 0,C 180,E1 -20186.01,E2 -20186.01} C_VEL
LIN {X 0,Y 284.985,Z 567.147,A -85,B 0,C 180,E1 -20186.559,E2 -20186.559} C_VEL
LIN {X 0,Y 288.913,Z 550.598,A -85,B 0,C 180,E1 -20187.381,E2 -20187.381} C_VEL
LIN {X 0,Y 300.89,Z 482.824,A -85,B 0,C 180,E1 -20189.734,E2 -20189.734} C_VEL
LIN {X 0,Y 300.23,Z 480.93,A -85,B 0,C 180,E1 -20190.828,E2 -20190.828} C_VEL
LIN {X 0,Y 299.504,Z 478.973,A -85,B 0,C 180,E1 -20192.477,E2 -20192.477} C_VEL
LIN {X 0,Y 299.007,Z 478.22,A -85,B 0,C 180,E1 -20194.34,E2 -20194.34} C_VEL
LIN {X 0,Y 298.899,Z 478.623,A -85,B 0,C 180,E1 -20196.002,E2 -20196.002} C_VEL
LIN {X 0,Y 299.396,Z 480.83,A -85,B 0,C 180,E1 -20198.471,E2 -20198.471} C_VEL
LIN {X 0,Y 300.182,Z 484.699,A -85,B 0,C 180,E1 -20200.421,E2 -20200.421} C_VEL
LIN {X 0,Y 300.466,Z 486.129,A -85,B 0,C 180,E1 -20200.996,E2 -20200.996} C_VEL
LIN {X 0,Y 288.367,Z 555.09,A -85,B 0,C 180,E1 -20203.397,E2 -20203.397} C_VEL
LIN {X 0,Y 284.741,Z 570.433,A -85,B 0,C 180,E1 -20204.094,E2 -20204.094} C_VEL
LIN {X 0,Y 280.285,Z 585.415,A -85,B 0,C 180,E1 -20204.966,E2 -20204.966} C_VEL
LIN {X 0,Y 274.952,Z 600.295,A -85,B 0,C 180,E1 -20206.103,E2 -20206.103} C_VEL
LIN {X 0,Y 268.628,Z 615.623,A -85,B 0,C 180,E1 -20207.645,E2 -20207.645} C_VEL
LIN {X 0,Y 262.647,Z 628.437,A -85,B 0,C 180,E1 -20209.287,E2 -20209.287} C_VEL
LIN {X 0,Y 256.071,Z 641.252,A -85,B 0,C 180,E1 -20211.36,E2 -20211.36} C_VEL
LIN {X 0,Y 249.523,Z 652.955,A -85,B 0,C 180,E1 -20213.735,E2 -20213.735} C_VEL
LIN {X 0,Y 242.731,Z 664.229,A -85,B 0,C 180,E1 -20216.622,E2 -20216.622} C_VEL
LIN {X 0,Y 236.745,Z 673.595,A -85,B 0,C 180,E1 -20219.689,E2 -20219.689} C_VEL
LIN {X 0,Y 231.749,Z 681.36,A -85,B 0,C 180,E1 -20222.94,E2 -20222.94} C_VEL
LIN {X 0,Y 227.535,Z 687.685,A -85,B 0,C 180,E1 -20226.323,E2 -20226.323} C_VEL
LIN {X 0,Y 223.993,Z 692.772,A -85,B 0,C 180,E1 -20229.807,E2 -20229.807} C_VEL
LIN {X 0,Y 221.476,Z 696.629,A -85,B 0,C 180,E1 -20233.403,E2 -20233.403} C_VEL
LIN {X 0,Y 219.749,Z 699.348,A -85,B 0,C 180,E1 -20237.061,E2 -20237.061} C_VEL
LIN {X 0,Y 218.837,Z 700.881,A -85,B 0,C 180,E1 -20240.757,E2 -20240.757} C_VEL
LIN {X 0,Y 218.479,Z 701.26,A -85,B 0,C 180,E1 -20244.459,E2 -20244.459} C_VEL
LIN {X 0,Y 218.617,Z 700.469,A -85,B 0,C 180,E1 -20248.155,E2 -20248.155} C_VEL
LIN {X 0,Y 218.716,Z 699.614,A -85,B 0,C 180,E1 -20249.997,E2 -20249.997} C_VEL
LIN {X 0,Y 218.726,Z 698.431,A -85,B 0,C 180,E1 -20251.839,E2 -20251.839} C_VEL
LIN {X 0,Y 218.727,Z 695.041,A -85,B 0,C 180,E1 -20255.529,E2 -20255.529} C_VEL
LIN {X 0,Y 218.908,Z 690.184,A -85,B 0,C 180,E1 -20259.234,E2 -20259.234} C_VEL
LIN {X 0,Y 219.559,Z 683.701,A -85,B 0,C 180,E1 -20262.945,E2 -20262.945} C_VEL
LIN {X 0,Y 220.651,Z 676.61,A -85,B 0,C 180,E1 -20266.179,E2 -20266.179} C_VEL
LIN {X 0,Y 222.268,Z 667.974,A -85,B 0,C 180,E1 -20269.387,E2 -20269.387} C_VEL
LIN {X 0,Y 224.472,Z 657.521,A -85,B 0,C 180,E1 -20272.55,E2 -20272.55} C_VEL
LIN {X 0,Y 226.703,Z 646.784,A -85,B 0,C 180,E1 -20275.227,E2 -20275.227} C_VEL
LIN {X 0,Y 229.296,Z 635.194,A -85,B 0,C 180,E1 -20277.615,E2 -20277.615} C_VEL
LIN {X 0,Y 231.853,Z 622.636,A -85,B 0,C 180,E1 -20279.756,E2 -20279.756} C_VEL
LIN {X 0,Y 234.447,Z 609.105,A -85,B 0,C 180,E1 -20281.638,E2 -20281.638} C_VEL
LIN {X 0,Y 237.02,Z 594.43,A -85,B 0,C 180,E1 -20283.264,E2 -20283.264} C_VEL
LIN {X 0,Y 239.207,Z 579.513,A -85,B 0,C 180,E1 -20284.558,E2 -20284.558} C_VEL
LIN {X 0,Y 241.138,Z 563.178,A -85,B 0,C 180,E1 -20285.604,E2 -20285.604} C_VEL
LIN {X 0,Y 242.628,Z 544.57,A -85,B 0,C 180,E1 -20286.424,E2 -20286.424} C_VEL
LIN {X 0,Y 249.032,Z 455.148,A -85,B 0,C 180,E1 -20289.824,E2 -20289.824} C_VEL
LIN {X 0,Y 239.71,Z 431.398,A -85,B 0,C 180,E1 -20292.13,E2 -20292.13} C_VEL
LIN {X 0,Y 230.857,Z 410.788,A -85,B 0,C 180,E1 -20294.456,E2 -20294.456} C_VEL
LIN {X 0,Y 221.629,Z 390.787,A -85,B 0,C 180,E1 -20297.047,E2 -20297.047} C_VEL
LIN {X 0,Y 220.734,Z 387.617,A -85,B 0,C 180,E1 -20298.405,E2 -20298.405} C_VEL
LIN {X 0,Y 220.814,Z 387.607,A -85,B 0,C 180,E1 -20302.791,E2 -20302.791} C_VEL
LIN {X 0,Y 220.799,Z 387.607,A -85,B 0,C 180,E1 -20307.242,E2 -20307.242} C_VEL
LIN {X 0,Y 220.783,Z 387.608,A -85,B 0,C 180,E1 -20311.479,E2 -20311.479} C_VEL
LIN {X 0,Y 220.79,Z 387.602,A -85,B 0,C 180,E1 -20315.556,E2 -20315.556} C_VEL
LIN {X 0,Y 220.834,Z 387.6,A -85,B 0,C 180,E1 -20319.509,E2 -20319.509} C_VEL
LIN {X 0,Y 220.957,Z 387.583,A -85,B 0,C 180,E1 -20323.366,E2 -20323.366} C_VEL
LIN {X 0,Y 221.037,Z 387.562,A -85,B 0,C 180,E1 -20329.003,E2 -20329.003} C_VEL
LIN {X 0,Y 221.222,Z 387.551,A -85,B 0,C 180,E1 -20332.7,E2 -20332.7} C_VEL
LIN {X 0,Y 221.454,Z 387.523,A -85,B 0,C 180,E1 -20338.182,E2 -20338.182} C_VEL
LIN {X 0,Y 221.454,Z 387.524,A -85,B 0,C 180,E1 -20341.819,E2 -20341.819} C_VEL
LIN {X 0,Y 221.228,Z 387.552,A -85,B 0,C 180,E1 -20347.301,E2 -20347.301} C_VEL
LIN {X 0,Y 221.037,Z 387.57,A -85,B 0,C 180,E1 -20350.998,E2 -20350.998} C_VEL
LIN {X 0,Y 220.958,Z 387.579,A -85,B 0,C 180,E1 -20356.635,E2 -20356.635} C_VEL
LIN {X 0,Y 220.835,Z 387.601,A -85,B 0,C 180,E1 -20360.492,E2 -20360.492} C_VEL
LIN {X 0,Y 220.792,Z 387.6,A -85,B 0,C 180,E1 -20364.445,E2 -20364.445} C_VEL
LIN {X 0,Y 220.785,Z 387.606,A -85,B 0,C 180,E1 -20368.522,E2 -20368.522} C_VEL
LIN {X 0,Y 220.801,Z 387.599,A -85,B 0,C 180,E1 -20372.759,E2 -20372.759} C_VEL
LIN {X 0,Y 220.791,Z 387.604,A -85,B 0,C 180,E1 -20377.277,E2 -20377.277} C_VEL
LIN {X 0,Y 220.746,Z 387.605,A -85,B 0,C 180,E1 -20381.959,E2 -20381.959} C_VEL
LIN {X 0,Y 220.746,Z 387.611,A -85,B 0,C 180,E1 -20385.543,E2 -20385.543} C_VEL
LIN {X 0,Y 220.774,Z 387.6,A -85,B 0,C 180,E1 -20390.46,E2 -20390.46} C_VEL
LIN {X 0,Y 220.819,Z 387.6,A -85,B 0,C 180,E1 -20392.796,E2 -20392.796} C_VEL
LIN {X 0,Y 220.806,Z 387.602,A -85,B 0,C 180,E1 -20397.246,E2 -20397.246} C_VEL
LIN {X 0,Y 220.792,Z 387.607,A -85,B 0,C 180,E1 -20401.484,E2 -20401.484} C_VEL
LIN {X 0,Y 220.804,Z 387.601,A -85,B 0,C 180,E1 -20405.561,E2 -20405.561} C_VEL
LIN {X 0,Y 220.869,Z 387.599,A -85,B 0,C 180,E1 -20409.515,E2 -20409.515} C_VEL
LIN {X 0,Y 220.979,Z 387.569,A -85,B 0,C 180,E1 -20413.37,E2 -20413.37} C_VEL
LIN {X 0,Y 221.005,Z 387.57,A -85,B 0,C 180,E1 -20417.141,E2 -20417.141} C_VEL
LIN {X 0,Y 221.195,Z 387.556,A -85,B 0,C 180,E1 -20420.862,E2 -20420.862} C_VEL
LIN {X 0,Y 221.112,Z 387.552,A -85,B 0,C 180,E1 -20424.531,E2 -20424.531} C_VEL
LIN {X 0,Y 221.472,Z 387.524,A -85,B 0,C 180,E1 -20428.184,E2 -20428.184} C_VEL
LIN {X 0,Y 221.472,Z 387.515,A -85,B 0,C 180,E1 -20431.821,E2 -20431.821} C_VEL
LIN {X 0,Y 221.244,Z 387.553,A -85,B 0,C 180,E1 -20437.303,E2 -20437.303} C_VEL
LIN {X 0,Y 221.065,Z 387.572,A -85,B 0,C 180,E1 -20440.999,E2 -20440.999} C_VEL
LIN {X 0,Y 220.976,Z 387.584,A -85,B 0,C 180,E1 -20446.636,E2 -20446.636} C_VEL
LIN {X 0,Y 220.881,Z 387.597,A -85,B 0,C 180,E1 -20450.49,E2 -20450.49} C_VEL
LIN {X 0,Y 220.839,Z 387.6,A -85,B 0,C 180,E1 -20454.441,E2 -20454.441} C_VEL
LIN {X 0,Y 221.866,Z 390.532,A -85,B 0,C 180,E1 -20454.819,E2 -20454.819} C_VEL
LIN {X 0,Y 224.793,Z 395.709,A -85,B 0,C 180,E1 -20455.587,E2 -20455.587} C_VEL
LIN {X 0,Y 234.687,Z 414.558,A -85,B 0,C 180,E1 -20458.072,E2 -20458.072} C_VEL
LIN {X 0,Y 242.778,Z 431.254,A -85,B 0,C 180,E1 -20460.021,E2 -20460.021} C_VEL
LIN {X 0,Y 248.894,Z 446.32,A -85,B 0,C 180,E1 -20461.496,E2 -20461.496} C_VEL
LIN {X 0,Y 241.746,Z 545.121,A -85,B 0,C 180,E1 -20465.285,E2 -20465.285} C_VEL
LIN {X 0,Y 240.088,Z 561.029,A -85,B 0,C 180,E1 -20466.212,E2 -20466.212} C_VEL
LIN {X 0,Y 238.126,Z 576.465,A -85,B 0,C 180,E1 -20467.451,E2 -20467.451} C_VEL
LIN {X 0,Y 235.821,Z 591.062,A -85,B 0,C 180,E1 -20468.958,E2 -20468.958} C_VEL
LIN {X 0,Y 233.257,Z 605.267,A -85,B 0,C 180,E1 -20470.798,E2 -20470.798} C_VEL
LIN {X 0,Y 230.548,Z 618.874,A -85,B 0,C 180,E1 -20472.977,E2 -20472.977} C_VEL
LIN {X 0,Y 227.905,Z 631.78,A -85,B 0,C 180,E1 -20475.522,E2 -20475.522} C_VEL
LIN {X 0,Y 225.401,Z 643.162,A -85,B 0,C 180,E1 -20478.249,E2 -20478.249} C_VEL
LIN {X 0,Y 223.432,Z 652.712,A -85,B 0,C 180,E1 -20481.016,E2 -20481.016} C_VEL
LIN {X 0,Y 221.627,Z 661.51,A -85,B 0,C 180,E1 -20484.079,E2 -20484.079} C_VEL
LIN {X 0,Y 220.165,Z 669.909,A -85,B 0,C 180,E1 -20487.677,E2 -20487.677} C_VEL
LIN {X 0,Y 219.222,Z 676.514,A -85,B 0,C 180,E1 -20491.256,E2 -20491.256} C_VEL
LIN {X 0,Y 218.67,Z 680.786,A -85,B 0,C 180,E1 -20494.151,E2 -20494.151} C_VEL
LIN {X 0,Y 218.234,Z 684.362,A -85,B 0,C 180,E1 -20497.266,E2 -20497.266} C_VEL
LIN {X 0,Y 218.155,Z 686.148,A -85,B 0,C 180,E1 -20499.244,E2 -20499.244} C_VEL
LIN {X 0,Y 218.194,Z 688.604,A -85,B 0,C 180,E1 -20503.148,E2 -20503.148} C_VEL
LIN {X 0,Y 218.679,Z 689.699,A -85,B 0,C 180,E1 -20506.998,E2 -20506.998} C_VEL
LIN {X 0,Y 219.648,Z 689.541,A -85,B 0,C 180,E1 -20510.794,E2 -20510.794} C_VEL
LIN {X 0,Y 221.258,Z 688.184,A -85,B 0,C 180,E1 -20514.531,E2 -20514.531} C_VEL
LIN {X 0,Y 223.574,Z 685.668,A -85,B 0,C 180,E1 -20518.198,E2 -20518.198} C_VEL
LIN {X 0,Y 226.647,Z 681.923,A -85,B 0,C 180,E1 -20521.776,E2 -20521.776} C_VEL
LIN {X 0,Y 230.505,Z 676.91,A -85,B 0,C 180,E1 -20525.248,E2 -20525.248} C_VEL
LIN {X 0,Y 235.191,Z 670.532,A -85,B 0,C 180,E1 -20528.592,E2 -20528.592} C_VEL
LIN {X 0,Y 240.751,Z 662.635,A -85,B 0,C 180,E1 -20531.791,E2 -20531.791} C_VEL
LIN {X 0,Y 246.178,Z 654.311,A -85,B 0,C 180,E1 -20534.465,E2 -20534.465} C_VEL
LIN {X 0,Y 252.267,Z 644.438,A -85,B 0,C 180,E1 -20537.009,E2 -20537.009} C_VEL
LIN {X 0,Y 257.911,Z 634.474,A -85,B 0,C 180,E1 -20539.086,E2 -20539.086} C_VEL
LIN {X 0,Y 264.024,Z 622.632,A -85,B 0,C 180,E1 -20541.111,E2 -20541.111} C_VEL
LIN {X 0,Y 270.285,Z 609.098,A -85,B 0,C 180,E1 -20542.956,E2 -20542.956} C_VEL
LIN {X 0,Y 276.497,Z 593.762,A -85,B 0,C 180,E1 -20544.596,E2 -20544.596} C_VEL
LIN {X 0,Y 281.937,Z 577.798,A -85,B 0,C 180,E1 -20545.885,E2 -20545.885} C_VEL
LIN {X 0,Y 284.985,Z 567.147,A -85,B 0,C 180,E1 -20546.559,E2 -20546.559} C_VEL
LIN {X 0,Y 285.738,Z 563.585,A -85,B 0,C 180,E1 -20546.899,E2 -20546.899} C_VEL
LIN {X 0,Y 286.735,Z 552.878,A -85,B 0,C 180,E1 -20548.54,E2 -20548.54} C_VEL
LIN {X 0,Y 287.311,Z 549.195,A -85,B 0,C 180,E1 -20548.807,E2 -20548.807} C_VEL
LIN {X 0,Y 298.596,Z 488.224,A -85,B 0,C 180,E1 -20550.887,E2 -20550.887} C_VEL
LIN {X 0,Y 298.641,Z 487.861,A -85,B 0,C 180,E1 -20550.924,E2 -20550.924} C_VEL
LIN {X 0,Y 297.923,Z 485.821,A -85,B 0,C 180,E1 -20552.671,E2 -20552.671} C_VEL
LIN {X 0,Y 297.534,Z 485.166,A -85,B 0,C 180,E1 -20554.233,E2 -20554.233} C_VEL
LIN {X 0,Y 297.392,Z 485.516,A -85,B 0,C 180,E1 -20555.851,E2 -20555.851} C_VEL
LIN {X 0,Y 297.726,Z 487.449,A -85,B 0,C 180,E1 -20558.062,E2 -20558.062} C_VEL
LIN {X 0,Y 298.261,Z 490.775,A -85,B 0,C 180,E1 -20559.809,E2 -20559.809} C_VEL
LIN {X 0,Y 286.279,Z 555.616,A -85,B 0,C 180,E1 -20562.047,E2 -20562.047} C_VEL
LIN {X 0,Y 282.657,Z 570.141,A -85,B 0,C 180,E1 -20562.687,E2 -20562.687} C_VEL
LIN {X 0,Y 277.782,Z 585.661,A -85,B 0,C 180,E1 -20563.593,E2 -20563.593} C_VEL
LIN {X 0,Y 272.697,Z 599.258,A -85,B 0,C 180,E1 -20564.603,E2 -20564.603} C_VEL
LIN {X 0,Y 266.665,Z 613.359,A -85,B 0,C 180,E1 -20565.961,E2 -20565.961} C_VEL
LIN {X 0,Y 260.377,Z 626.285,A -85,B 0,C 180,E1 -20567.56,E2 -20567.56} C_VEL
LIN {X 0,Y 253.867,Z 638.467,A -85,B 0,C 180,E1 -20569.413,E2 -20569.413} C_VEL
LIN {X 0,Y 246.868,Z 650.392,A -85,B 0,C 180,E1 -20571.74,E2 -20571.74} C_VEL
LIN {X 0,Y 240.467,Z 660.634,A -85,B 0,C 180,E1 -20574.228,E2 -20574.228} C_VEL
LIN {X 0,Y 235.412,Z 668.141,A -85,B 0,C 180,E1 -20576.472,E2 -20576.472} C_VEL
LIN {X 0,Y 230.732,Z 674.802,A -85,B 0,C 180,E1 -20578.812,E2 -20578.812} C_VEL
LIN {X 0,Y 225.502,Z 682.24,A -85,B 0,C 180,E1 -20582.126,E2 -20582.126} C_VEL
LIN {X 0,Y 221.063,Z 688.373,A -85,B 0,C 180,E1 -20585.585,E2 -20585.585} C_VEL
LIN {X 0,Y 217.331,Z 693.189,A -85,B 0,C 180,E1 -20589.16,E2 -20589.16} C_VEL
LIN {X 0,Y 214.618,Z 696.841,A -85,B 0,C 180,E1 -20592.857,E2 -20592.857} C_VEL
LIN {X 0,Y 212.782,Z 699.352,A -85,B 0,C 180,E1 -20596.629,E2 -20596.629} C_VEL
LIN {X 0,Y 211.793,Z 700.764,A -85,B 0,C 180,E1 -20600.447,E2 -20600.447} C_VEL
LIN {X 0,Y 211.385,Z 700.994,A -85,B 0,C 180,E1 -20604.273,E2 -20604.273} C_VEL
LIN {X 0,Y 211.529,Z 700.046,A -85,B 0,C 180,E1 -20608.093,E2 -20608.093} C_VEL
LIN {X 0,Y 211.651,Z 699.109,A -85,B 0,C 180,E1 -20609.997,E2 -20609.997} C_VEL
LIN {X 0,Y 211.661,Z 697.841,A -85,B 0,C 180,E1 -20611.9,E2 -20611.9} C_VEL
LIN {X 0,Y 211.641,Z 694.268,A -85,B 0,C 180,E1 -20615.714,E2 -20615.714} C_VEL
LIN {X 0,Y 211.875,Z 689.221,A -85,B 0,C 180,E1 -20619.544,E2 -20619.544} C_VEL
LIN {X 0,Y 212.587,Z 682.559,A -85,B 0,C 180,E1 -20623.377,E2 -20623.377} C_VEL
LIN {X 0,Y 213.77,Z 675.284,A -85,B 0,C 180,E1 -20626.715,E2 -20626.715} C_VEL
LIN {X 0,Y 215.499,Z 666.444,A -85,B 0,C 180,E1 -20630.022,E2 -20630.022} C_VEL
LIN {X 0,Y 217.443,Z 657.415,A -85,B 0,C 180,E1 -20632.818,E2 -20632.818} C_VEL
LIN {X 0,Y 219.737,Z 646.688,A -85,B 0,C 180,E1 -20635.577,E2 -20635.577} C_VEL
LIN {X 0,Y 222.606,Z 633.9,A -85,B 0,C 180,E1 -20638.263,E2 -20638.263} C_VEL
LIN {X 0,Y 225.303,Z 621.146,A -85,B 0,C 180,E1 -20640.454,E2 -20640.454} C_VEL
LIN {X 0,Y 228,Z 607.343,A -85,B 0,C 180,E1 -20642.379,E2 -20642.379} C_VEL
LIN {X 0,Y 230.658,Z 592.299,A -85,B 0,C 180,E1 -20644.043,E2 -20644.043} C_VEL
LIN {X 0,Y 233,Z 576.475,A -85,B 0,C 180,E1 -20645.39,E2 -20645.39} C_VEL
LIN {X 0,Y 234.91,Z 560.089,A -85,B 0,C 180,E1 -20646.407,E2 -20646.407} C_VEL
LIN {X 0,Y 237.134,Z 529.786,A -85,B 0,C 180,E1 -20647.678,E2 -20647.678} C_VEL
LIN {X 0,Y 242.577,Z 456.741,A -85,B 0,C 180,E1 -20650.529,E2 -20650.529} C_VEL
LIN {X 0,Y 232.773,Z 431.596,A -85,B 0,C 180,E1 -20653.091,E2 -20653.091} C_VEL
LIN {X 0,Y 222.819,Z 409.056,A -85,B 0,C 180,E1 -20655.774,E2 -20655.774} C_VEL
LIN {X 0,Y 215.656,Z 393.834,A -85,B 0,C 180,E1 -20657.846,E2 -20657.846} C_VEL
LIN {X 0,Y 214.216,Z 390.514,A -85,B 0,C 180,E1 -20658.367,E2 -20658.367} C_VEL
LIN {X 0,Y 213.707,Z 388.492,A -85,B 0,C 180,E1 -20659.302,E2 -20659.302} C_VEL
LIN {X 0,Y 213.73,Z 388.49,A -85,B 0,C 180,E1 -20663.71,E2 -20663.71} C_VEL
LIN {X 0,Y 213.747,Z 388.487,A -85,B 0,C 180,E1 -20668.26,E2 -20668.26} C_VEL
LIN {X 0,Y 213.771,Z 388.479,A -85,B 0,C 180,E1 -20672.596,E2 -20672.596} C_VEL
LIN {X 0,Y 213.782,Z 388.481,A -85,B 0,C 180,E1 -20676.989,E2 -20676.989} C_VEL
LIN {X 0,Y 213.866,Z 388.467,A -85,B 0,C 180,E1 -20682.798,E2 -20682.798} C_VEL
LIN {X 0,Y 213.901,Z 388.462,A -85,B 0,C 180,E1 -20686.704,E2 -20686.704} C_VEL
LIN {X 0,Y 214.115,Z 388.426,A -85,B 0,C 180,E1 -20690.555,E2 -20690.555} C_VEL
LIN {X 0,Y 214.06,Z 388.446,A -85,B 0,C 180,E1 -20694.348,E2 -20694.348} C_VEL
LIN {X 0,Y 214.391,Z 388.402,A -85,B 0,C 180,E1 -20698.122,E2 -20698.122} C_VEL
LIN {X 0,Y 214.499,Z 388.393,A -85,B 0,C 180,E1 -20700.001,E2 -20700.001} C_VEL
LIN {X 0,Y 214.39,Z 388.403,A -85,B 0,C 180,E1 -20701.879,E2 -20701.879} C_VEL
LIN {X 0,Y 214.17,Z 388.432,A -85,B 0,C 180,E1 -20707.543,E2 -20707.543} C_VEL
LIN {X 0,Y 213.97,Z 388.451,A -85,B 0,C 180,E1 -20711.366,E2 -20711.366} C_VEL
LIN {X 0,Y 213.86,Z 388.469,A -85,B 0,C 180,E1 -20715.243,E2 -20715.243} C_VEL
LIN {X 0,Y 213.779,Z 388.475,A -85,B 0,C 180,E1 -20719.194,E2 -20719.194} C_VEL
LIN {X 0,Y 213.773,Z 388.479,A -85,B 0,C 180,E1 -20723.236,E2 -20723.236} C_VEL
LIN {X 0,Y 213.775,Z 388.476,A -85,B 0,C 180,E1 -20727.429,E2 -20727.429} C_VEL
LIN {X 0,Y 213.749,Z 388.483,A -85,B 0,C 180,E1 -20731.741,E2 -20731.741} C_VEL
LIN {X 0,Y 213.732,Z 388.484,A -85,B 0,C 180,E1 -20736.291,E2 -20736.291} C_VEL
LIN {X 0,Y 213.693,Z 388.486,A -85,B 0,C 180,E1 -20741.131,E2 -20741.131} C_VEL
LIN {X 0,Y 213.694,Z 388.484,A -85,B 0,C 180,E1 -20743.682,E2 -20743.682} C_VEL
LIN {X 0,Y 213.694,Z 388.49,A -85,B 0,C 180,E1 -20746.348,E2 -20746.348} C_VEL
LIN {X 0,Y 213.695,Z 388.482,A -85,B 0,C 180,E1 -20751.331,E2 -20751.331} C_VEL
LIN {X 0,Y 213.748,Z 388.483,A -85,B 0,C 180,E1 -20756.02,E2 -20756.02} C_VEL
LIN {X 0,Y 213.743,Z 388.483,A -85,B 0,C 180,E1 -20760.452,E2 -20760.452} C_VEL
LIN {X 0,Y 213.749,Z 388.479,A -85,B 0,C 180,E1 -20764.699,E2 -20764.699} C_VEL
LIN {X 0,Y 213.788,Z 388.479,A -85,B 0,C 180,E1 -20768.804,E2 -20768.804} C_VEL
LIN {X 0,Y 213.893,Z 388.456,A -85,B 0,C 180,E1 -20772.803,E2 -20772.803} C_VEL
LIN {X 0,Y 213.943,Z 388.449,A -85,B 0,C 180,E1 -20776.709,E2 -20776.709} C_VEL
LIN {X 0,Y 214.135,Z 388.435,A -85,B 0,C 180,E1 -20780.558,E2 -20780.558} C_VEL
LIN {X 0,Y 214.075,Z 388.428,A -85,B 0,C 180,E1 -20784.351,E2 -20784.351} C_VEL
LIN {X 0,Y 214.409,Z 388.404,A -85,B 0,C 180,E1 -20788.124,E2 -20788.124} C_VEL
LIN {X 0,Y 214.516,Z 388.389,A -85,B 0,C 180,E1 -20790.003,E2 -20790.003} C_VEL
LIN {X 0,Y 214.409,Z 388.394,A -85,B 0,C 180,E1 -20791.881,E2 -20791.881} C_VEL
LIN {X 0,Y 214.186,Z 388.43,A -85,B 0,C 180,E1 -20797.545,E2 -20797.545} C_VEL
LIN {X 0,Y 213.994,Z 388.454,A -85,B 0,C 180,E1 -20801.367,E2 -20801.367} C_VEL
LIN {X 0,Y 213.879,Z 388.464,A -85,B 0,C 180,E1 -20805.244,E2 -20805.244} C_VEL
LIN {X 0,Y 213.812,Z 388.474,A -85,B 0,C 180,E1 -20809.193,E2 -20809.193} C_VEL
LIN {X 0,Y 213.789,Z 388.494,A -85,B 0,C 180,E1 -20813.308,E2 -20813.308} C_VEL
LIN {X 0,Y 214.744,Z 391.268,A -85,B 0,C 180,E1 -20813.637,E2 -20813.637} C_VEL
LIN {X 0,Y 216.068,Z 393.491,A -85,B 0,C 180,E1 -20813.992,E2 -20813.992} C_VEL
LIN {X 0,Y 225,Z 410.126,A -85,B 0,C 180,E1 -20816.402,E2 -20816.402} C_VEL
LIN {X 0,Y 234.522,Z 429.128,A -85,B 0,C 180,E1 -20818.79,E2 -20818.79} C_VEL
LIN {X 0,Y 238.89,Z 439.027,A -85,B 0,C 180,E1 -20819.884,E2 -20819.884} C_VEL
LIN {X 0,Y 242.526,Z 448.105,A -85,B 0,C 180,E1 -20820.798,E2 -20820.798} C_VEL
LIN {X 0,Y 235.167,Z 545.726,A -85,B 0,C 180,E1 -20824.646,E2 -20824.646} C_VEL
LIN {X 0,Y 233.422,Z 561.778,A -85,B 0,C 180,E1 -20825.616,E2 -20825.616} C_VEL
LIN {X 0,Y 231.337,Z 577.522,A -85,B 0,C 180,E1 -20826.929,E2 -20826.929} C_VEL
LIN {X 0,Y 228.969,Z 592.068,A -85,B 0,C 180,E1 -20828.49,E2 -20828.49} C_VEL
LIN {X 0,Y 226.33,Z 606.308,A -85,B 0,C 180,E1 -20830.408,E2 -20830.408} C_VEL
LIN {X 0,Y 223.51,Z 620.015,A -85,B 0,C 180,E1 -20832.692,E2 -20832.692} C_VEL
LIN {X 0,Y 221.048,Z 631.603,A -85,B 0,C 180,E1 -20835.051,E2 -20835.051} C_VEL
LIN {X 0,Y 218.628,Z 642.35,A -85,B 0,C 180,E1 -20837.68,E2 -20837.68} C_VEL
LIN {X 0,Y 216.52,Z 652.164,A -85,B 0,C 180,E1 -20840.566,E2 -20840.566} C_VEL
LIN {X 0,Y 214.596,Z 661.452,A -85,B 0,C 180,E1 -20843.878,E2 -20843.878} C_VEL
LIN {X 0,Y 213.265,Z 668.798,A -85,B 0,C 180,E1 -20847.06,E2 -20847.06} C_VEL
LIN {X 0,Y 212.328,Z 674.841,A -85,B 0,C 180,E1 -20850.231,E2 -20850.231} C_VEL
LIN {X 0,Y 211.65,Z 680.117,A -85,B 0,C 180,E1 -20853.714,E2 -20853.714} C_VEL
LIN {X 0,Y 211.245,Z 683.429,A -85,B 0,C 180,E1 -20856.469,E2 -20856.469} C_VEL
LIN {X 0,Y 211.022,Z 687.039,A -85,B 0,C 180,E1 -20860.546,E2 -20860.546} C_VEL
LIN {X 0,Y 211.238,Z 689.198,A -85,B 0,C 180,E1 -20864.563,E2 -20864.563} C_VEL
LIN {X 0,Y 211.888,Z 690.052,A -85,B 0,C 180,E1 -20868.52,E2 -20868.52} C_VEL
LIN {X 0,Y 213.212,Z 689.634,A -85,B 0,C 180,E1 -20872.423,E2 -20872.423} C_VEL
LIN {X 0,Y 215.092,Z 688.056,A -85,B 0,C 180,E1 -20876.253,E2 -20876.253} C_VEL
LIN {X 0,Y 217.876,Z 685.206,A -85,B 0,C 180,E1 -20880.098,E2 -20880.098} C_VEL
LIN {X 0,Y 221.362,Z 681.362,A -85,B 0,C 180,E1 -20883.64,E2 -20883.64} C_VEL
LIN {X 0,Y 225.728,Z 676.146,A -85,B 0,C 180,E1 -20887.154,E2 -20887.154} C_VEL
LIN {X 0,Y 230.958,Z 669.587,A -85,B 0,C 180,E1 -20890.52,E2 -20890.52} C_VEL
LIN {X 0,Y 237.02,Z 661.415,A -85,B 0,C 180,E1 -20893.722,E2 -20893.722} C_VEL
LIN {X 0,Y 242.791,Z 653.173,A -85,B 0,C 180,E1 -20896.318,E2 -20896.318} C_VEL
LIN {X 0,Y 249.467,Z 642.777,A -85,B 0,C 180,E1 -20898.903,E2 -20898.903} C_VEL
LIN {X 0,Y 256.316,Z 631.187,A -85,B 0,C 180,E1 -20901.206,E2 -20901.206} C_VEL
LIN {X 0,Y 263.039,Z 618.416,A -85,B 0,C 180,E1 -20903.209,E2 -20903.209} C_VEL
LIN {X 0,Y 269.325,Z 605.087,A -85,B 0,C 180,E1 -20904.884,E2 -20904.884} C_VEL
LIN {X 0,Y 274.637,Z 592.094,A -85,B 0,C 180,E1 -20906.177,E2 -20906.177} C_VEL
LIN {X 0,Y 280.341,Z 575.888,A -85,B 0,C 180,E1 -20907.429,E2 -20907.429} C_VEL
LIN {X 0,Y 284.623,Z 560.936,A -85,B 0,C 180,E1 -20908.28,E2 -20908.28} C_VEL
LIN {X 0,Y 287.311,Z 549.195,A -85,B 0,C 180,E1 -20908.807,E2 -20908.807} C_VEL
LIN {X 0,Y 288.261,Z 543.592,A -85,B 0,C 180,E1 -20909.127,E2 -20909.127} C_VEL
LIN {X 0,Y 290.412,Z 525.924,A -85,B 0,C 180,E1 -20910.868,E2 -20910.868} C_VEL
LIN {X 0,Y 291.355,Z 520.317,A -85,B 0,C 180,E1 -20911.187,E2 -20911.187} C_VEL
LIN {X 0,Y 296.603,Z 493.468,A -85,B 0,C 180,E1 -20912.096,E2 -20912.096} C_VEL
LIN {X 0,Y 296.193,Z 492.346,A -85,B 0,C 180,E1 -20913.355,E2 -20913.355} C_VEL
LIN {X 0,Y 295.879,Z 492.191,A -85,B 0,C 180,E1 -20915.295,E2 -20915.295} C_VEL
LIN {X 0,Y 296.078,Z 494.064,A -85,B 0,C 180,E1 -20917.664,E2 -20917.664} C_VEL
LIN {X 0,Y 296.271,Z 495.742,A -85,B 0,C 180,E1 -20918.614,E2 -20918.614} C_VEL
LIN {X 0,Y 284.784,Z 555.109,A -85,B 0,C 180,E1 -20920.634,E2 -20920.634} C_VEL
LIN {X 0,Y 280.677,Z 570.613,A -85,B 0,C 180,E1 -20921.305,E2 -20921.305} C_VEL
LIN {X 0,Y 275.293,Z 586.811,A -85,B 0,C 180,E1 -20922.237,E2 -20922.237} C_VEL
LIN {X 0,Y 270.04,Z 600.1,A -85,B 0,C 180,E1 -20923.218,E2 -20923.218} C_VEL
LIN {X 0,Y 263.794,Z 613.781,A -85,B 0,C 180,E1 -20924.545,E2 -20924.545} C_VEL
LIN {X 0,Y 257.239,Z 626.616,A -85,B 0,C 180,E1 -20926.108,E2 -20926.108} C_VEL
LIN {X 0,Y 250.968,Z 637.64,A -85,B 0,C 180,E1 -20927.769,E2 -20927.769} C_VEL
LIN {X 0,Y 243.591,Z 649.61,A -85,B 0,C 180,E1 -20930.06,E2 -20930.06} C_VEL
LIN {X 0,Y 236.764,Z 659.79,A -85,B 0,C 180,E1 -20932.515,E2 -20932.515} C_VEL
LIN {X 0,Y 230.463,Z 668.559,A -85,B 0,C 180,E1 -20935.123,E2 -20935.123} C_VEL
LIN {X 0,Y 224.784,Z 675.986,A -85,B 0,C 180,E1 -20937.889,E2 -20937.889} C_VEL
LIN {X 0,Y 219.303,Z 683.14,A -85,B 0,C 180,E1 -20941.266,E2 -20941.266} C_VEL
LIN {X 0,Y 214.634,Z 688.961,A -85,B 0,C 180,E1 -20944.804,E2 -20944.804} C_VEL
LIN {X 0,Y 210.689,Z 693.628,A -85,B 0,C 180,E1 -20948.471,E2 -20948.471} C_VEL
LIN {X 0,Y 207.785,Z 697.062,A -85,B 0,C 180,E1 -20952.274,E2 -20952.274} C_VEL
LIN {X 0,Y 205.833,Z 699.371,A -85,B 0,C 180,E1 -20956.169,E2 -20956.169} C_VEL
LIN {X 0,Y 204.769,Z 700.587,A -85,B 0,C 180,E1 -20960.116,E2 -20960.116} C_VEL
LIN {X 0,Y 204.319,Z 700.695,A -85,B 0,C 180,E1 -20964.074,E2 -20964.074} C_VEL
LIN {X 0,Y 204.444,Z 699.599,A -85,B 0,C 180,E1 -20968.027,E2 -20968.027} C_VEL
LIN {X 0,Y 204.587,Z 698.584,A -85,B 0,C 180,E1 -20969.997,E2 -20969.997} C_VEL
LIN {X 0,Y 204.598,Z 697.239,A -85,B 0,C 180,E1 -20971.966,E2 -20971.966} C_VEL
LIN {X 0,Y 204.562,Z 693.493,A -85,B 0,C 180,E1 -20975.913,E2 -20975.913} C_VEL
LIN {X 0,Y 204.817,Z 688.247,A -85,B 0,C 180,E1 -20979.876,E2 -20979.876} C_VEL
LIN {X 0,Y 205.63,Z 681.377,A -85,B 0,C 180,E1 -20983.839,E2 -20983.839} C_VEL
LIN {X 0,Y 206.901,Z 673.871,A -85,B 0,C 180,E1 -20987.287,E2 -20987.287} C_VEL
LIN {X 0,Y 208.756,Z 664.773,A -85,B 0,C 180,E1 -20990.698,E2 -20990.698} C_VEL
LIN {X 0,Y 211.22,Z 653.777,A -85,B 0,C 180,E1 -20994.051,E2 -20994.051} C_VEL
LIN {X 0,Y 213.708,Z 642.427,A -85,B 0,C 180,E1 -20996.88,E2 -20996.88} C_VEL
LIN {X 0,Y 216.532,Z 630.11,A -85,B 0,C 180,E1 -20999.397,E2 -20999.397} C_VEL
LIN {X 0,Y 219.372,Z 616.687,A -85,B 0,C 180,E1 -21001.638,E2 -21001.638} C_VEL
LIN {X 0,Y 222.278,Z 602.083,A -85,B 0,C 180,E1 -21003.591,E2 -21003.591} C_VEL
LIN {X 0,Y 224.866,Z 586.886,A -85,B 0,C 180,E1 -21005.183,E2 -21005.183} C_VEL
LIN {X 0,Y 227.088,Z 571.216,A -85,B 0,C 180,E1 -21006.423,E2 -21006.423} C_VEL
LIN {X 0,Y 228.856,Z 554.895,A -85,B 0,C 180,E1 -21007.348,E2 -21007.348} C_VEL
LIN {X 0,Y 236.242,Z 458.941,A -85,B 0,C 180,E1 -21011.226,E2 -21011.226} C_VEL
LIN {X 0,Y 228.959,Z 439.672,A -85,B 0,C 180,E1 -21013.216,E2 -21013.216} C_VEL
LIN {X 0,Y 219.898,Z 418.302,A -85,B 0,C 180,E1 -21015.723,E2 -21015.723} C_VEL
LIN {X 0,Y 210.713,Z 398.421,A -85,B 0,C 180,E1 -21018.446,E2 -21018.446} C_VEL
LIN {X 0,Y 206.906,Z 390.507,A -85,B 0,C 180,E1 -21019.638,E2 -21019.638} C_VEL
LIN {X 0,Y 206.709,Z 389.366,A -85,B 0,C 180,E1 -21020.234,E2 -21020.234} C_VEL
LIN {X 0,Y 206.688,Z 389.367,A -85,B 0,C 180,E1 -21024.687,E2 -21024.687} C_VEL
LIN {X 0,Y 206.682,Z 389.365,A -85,B 0,C 180,E1 -21029.333,E2 -21029.333} C_VEL
LIN {X 0,Y 206.673,Z 389.358,A -85,B 0,C 180,E1 -21033.764,E2 -21033.764} C_VEL
LIN {X 0,Y 206.701,Z 389.365,A -85,B 0,C 180,E1 -21038.037,E2 -21038.037} C_VEL
LIN {X 0,Y 206.79,Z 389.342,A -85,B 0,C 180,E1 -21042.19,E2 -21042.19} C_VEL
LIN {X 0,Y 206.842,Z 389.343,A -85,B 0,C 180,E1 -21046.241,E2 -21046.241} C_VEL
LIN {X 0,Y 207.06,Z 389.301,A -85,B 0,C 180,E1 -21050.23,E2 -21050.23} C_VEL
LIN {X 0,Y 207.023,Z 389.324,A -85,B 0,C 180,E1 -21054.155,E2 -21054.155} C_VEL
LIN {X 0,Y 207.33,Z 389.281,A -85,B 0,C 180,E1 -21058.058,E2 -21058.058} C_VEL
LIN {X 0,Y 207.467,Z 389.269,A -85,B 0,C 180,E1 -21060.001,E2 -21060.001} C_VEL
LIN {X 0,Y 207.33,Z 389.282,A -85,B 0,C 180,E1 -21061.943,E2 -21061.943} C_VEL
LIN {X 0,Y 207.114,Z 389.312,A -85,B 0,C 180,E1 -21067.802,E2 -21067.802} C_VEL
LIN {X 0,Y 206.891,Z 389.335,A -85,B 0,C 180,E1 -21071.761,E2 -21071.761} C_VEL
LIN {X 0,Y 206.793,Z 389.348,A -85,B 0,C 180,E1 -21075.777,E2 -21075.777} C_VEL
LIN {X 0,Y 206.7,Z 389.36,A -85,B 0,C 180,E1 -21079.878,E2 -21079.878} C_VEL
LIN {X 0,Y 206.69,Z 389.358,A -85,B 0,C 180,E1 -21084.082,E2 -21084.082} C_VEL
LIN {X 0,Y 206.676,Z 389.364,A -85,B 0,C 180,E1 -21088.43,E2 -21088.43} C_VEL
LIN {X 0,Y 206.684,Z 389.357,A -85,B 0,C 180,E1 -21092.961,E2 -21092.961} C_VEL
LIN {X 0,Y 206.659,Z 389.367,A -85,B 0,C 180,E1 -21097.745,E2 -21097.745} C_VEL
LIN {X 0,Y 206.625,Z 389.365,A -85,B 0,C 180,E1 -21101.563,E2 -21101.563} C_VEL
LIN {X 0,Y 206.622,Z 389.37,A -85,B 0,C 180,E1 -21105.586,E2 -21105.586} C_VEL
LIN {X 0,Y 206.639,Z 389.363,A -85,B 0,C 180,E1 -21109.748,E2 -21109.748} C_VEL
LIN {X 0,Y 206.695,Z 389.362,A -85,B 0,C 180,E1 -21114.692,E2 -21114.692} C_VEL
LIN {X 0,Y 206.69,Z 389.356,A -85,B 0,C 180,E1 -21119.337,E2 -21119.337} C_VEL
LIN {X 0,Y 206.684,Z 389.363,A -85,B 0,C 180,E1 -21123.769,E2 -21123.769} C_VEL
LIN {X 0,Y 206.724,Z 389.361,A -85,B 0,C 180,E1 -21128.043,E2 -21128.043} C_VEL
LIN {X 0,Y 206.825,Z 389.337,A -85,B 0,C 180,E1 -21132.196,E2 -21132.196} C_VEL
LIN {X 0,Y 206.883,Z 389.321,A -85,B 0,C 180,E1 -21136.247,E2 -21136.247} C_VEL
LIN {X 0,Y 207.08,Z 389.315,A -85,B 0,C 180,E1 -21140.233,E2 -21140.233} C_VEL
LIN {X 0,Y 207.039,Z 389.304,A -85,B 0,C 180,E1 -21144.158,E2 -21144.158} C_VEL
LIN {X 0,Y 207.348,Z 389.284,A -85,B 0,C 180,E1 -21148.061,E2 -21148.061} C_VEL
LIN {X 0,Y 207.484,Z 389.265,A -85,B 0,C 180,E1 -21150.003,E2 -21150.003} C_VEL
LIN {X 0,Y 207.348,Z 389.272,A -85,B 0,C 180,E1 -21151.945,E2 -21151.945} C_VEL
LIN {X 0,Y 207.131,Z 389.307,A -85,B 0,C 180,E1 -21157.803,E2 -21157.803} C_VEL
LIN {X 0,Y 206.914,Z 389.338,A -85,B 0,C 180,E1 -21161.762,E2 -21161.762} C_VEL
LIN {X 0,Y 206.813,Z 389.348,A -85,B 0,C 180,E1 -21165.778,E2 -21165.778} C_VEL
LIN {X 0,Y 206.75,Z 389.358,A -85,B 0,C 180,E1 -21169.875,E2 -21169.875} C_VEL
LIN {X 0,Y 206.746,Z 389.353,A -85,B 0,C 180,E1 -21172.074,E2 -21172.074} C_VEL
LIN {X 0,Y 207.761,Z 392.209,A -85,B 0,C 180,E1 -21172.45,E2 -21172.45} C_VEL
LIN {X 0,Y 209.38,Z 395.076,A -85,B 0,C 180,E1 -21172.921,E2 -21172.921} C_VEL
LIN {X 0,Y 218.149,Z 411.224,A -85,B 0,C 180,E1 -21175.367,E2 -21175.367} C_VEL
LIN {X 0,Y 228.503,Z 431.838,A -85,B 0,C 180,E1 -21178.082,E2 -21178.082} C_VEL
LIN {X 0,Y 233.072,Z 442.15,A -85,B 0,C 180,E1 -21179.25,E2 -21179.25} C_VEL
LIN {X 0,Y 236.156,Z 449.913,A -85,B 0,C 180,E1 -21180.062,E2 -21180.062} C_VEL
LIN {X 0,Y 228.704,Z 545.562,A -85,B 0,C 180,E1 -21183.931,E2 -21183.931} C_VEL
LIN {X 0,Y 227.003,Z 560.894,A -85,B 0,C 180,E1 -21184.87,E2 -21184.87} C_VEL
LIN {X 0,Y 224.769,Z 577.251,A -85,B 0,C 180,E1 -21186.259,E2 -21186.259} C_VEL
LIN {X 0,Y 222.198,Z 592.536,A -85,B 0,C 180,E1 -21187.948,E2 -21187.948} C_VEL
LIN {X 0,Y 219.626,Z 606.073,A -85,B 0,C 180,E1 -21189.825,E2 -21189.825} C_VEL
LIN {X 0,Y 216.826,Z 619.276,A -85,B 0,C 180,E1 -21192.071,E2 -21192.071} C_VEL
LIN {X 0,Y 214.014,Z 632.106,A -85,B 0,C 180,E1 -21194.753,E2 -21194.753} C_VEL
LIN {X 0,Y 211.327,Z 643.829,A -85,B 0,C 180,E1 -21197.746,E2 -21197.746} C_VEL
LIN {X 0,Y 209.052,Z 654.275,A -85,B 0,C 180,E1 -21201.01,E2 -21201.01} C_VEL
LIN {X 0,Y 207.17,Z 663.421,A -85,B 0,C 180,E1 -21204.509,E2 -21204.509} C_VEL
LIN {X 0,Y 205.883,Z 670.651,A -85,B 0,C 180,E1 -21207.906,E2 -21207.906} C_VEL
LIN {X 0,Y 205.005,Z 676.568,A -85,B 0,C 180,E1 -21211.317,E2 -21211.317} C_VEL
LIN {X 0,Y 204.405,Z 681.093,A -85,B 0,C 180,E1 -21214.546,E2 -21214.546} C_VEL
LIN {X 0,Y 203.958,Z 685.282,A -85,B 0,C 180,E1 -21218.499,E2 -21218.499} C_VEL
LIN {X 0,Y 203.944,Z 687.816,A -85,B 0,C 180,E1 -21221.931,E2 -21221.931} C_VEL
LIN {X 0,Y 204.304,Z 689.691,A -85,B 0,C 180,E1 -21226.066,E2 -21226.066} C_VEL
LIN {X 0,Y 205.212,Z 690.289,A -85,B 0,C 180,E1 -21230.14,E2 -21230.14} C_VEL
LIN {X 0,Y 206.822,Z 689.694,A -85,B 0,C 180,E1 -21234.148,E2 -21234.148} C_VEL
LIN {X 0,Y 209.138,Z 687.936,A -85,B 0,C 180,E1 -21238.074,E2 -21238.074} C_VEL
LIN {X 0,Y 212.317,Z 684.981,A -85,B 0,C 180,E1 -21241.896,E2 -21241.896} C_VEL
LIN {X 0,Y 216.355,Z 680.814,A -85,B 0,C 180,E1 -21245.592,E2 -21245.592} C_VEL
LIN {X 0,Y 221.234,Z 675.437,A -85,B 0,C 180,E1 -21249.139,E2 -21249.139} C_VEL
LIN {X 0,Y 226.985,Z 668.64,A -85,B 0,C 180,E1 -21252.517,E2 -21252.517} C_VEL
LIN {X 0,Y 233.628,Z 660.306,A -85,B 0,C 180,E1 -21255.708,E2 -21255.708} C_VEL
LIN {X 0,Y 241.034,Z 650.175,A -85,B 0,C 180,E1 -21258.707,E2 -21258.707} C_VEL
LIN {X 0,Y 247.072,Z 641.186,A -85,B 0,C 180,E1 -21260.828,E2 -21260.828} C_VEL
LIN {X 0,Y 254.642,Z 628.832,A -85,B 0,C 180,E1 -21263.159,E2 -21263.159} C_VEL
LIN {X 0,Y 261.524,Z 616.226,A -85,B 0,C 180,E1 -21265.04,E2 -21265.04} C_VEL
LIN {X 0,Y 268.27,Z 602.295,A -85,B 0,C 180,E1 -21266.682,E2 -21266.682} C_VEL
LIN {X 0,Y 273.287,Z 590.408,A -85,B 0,C 180,E1 -21267.782,E2 -21267.782} C_VEL
LIN {X 0,Y 278.828,Z 574.944,A -85,B 0,C 180,E1 -21268.922,E2 -21268.922} C_VEL
LIN {X 0,Y 282.963,Z 561.122,A -85,B 0,C 180,E1 -21269.682,E2 -21269.682} C_VEL
LIN {X 0,Y 286.379,Z 546.556,A -85,B 0,C 180,E1 -21270.294,E2 -21270.294} C_VEL
LIN {X 0,Y 291.355,Z 520.317,A -85,B 0,C 180,E1 -21271.187,E2 -21271.187} C_VEL
LIN {X 0,Y 291.989,Z 516.607,A -85,B 0,C 180,E1 -21271.446,E2 -21271.446} C_VEL
LIN {X 0,Y 293.525,Z 505.581,A -85,B 0,C 180,E1 -21272.947,E2 -21272.947} C_VEL
LIN {X 0,Y 294.204,Z 501.868,A -85,B 0,C 180,E1 -21273.194,E2 -21273.194} C_VEL
LIN {X 0,Y 294.701,Z 499.402,A -85,B 0,C 180,E1 -21273.264,E2 -21273.264} C_VEL
LIN {X 0,Y 294.393,Z 499.229,A -85,B 0,C 180,E1 -21275.5,E2 -21275.5} C_VEL
LIN {X 0,Y 294.451,Z 501.015,A -85,B 0,C 180,E1 -21277.417,E2 -21277.417} C_VEL
LIN {X 0,Y 283.639,Z 554.495,A -85,B 0,C 180,E1 -21279.185,E2 -21279.185} C_VEL
LIN {X 0,Y 278.896,Z 571.609,A -85,B 0,C 180,E1 -21279.912,E2 -21279.912} C_VEL
LIN {X 0,Y 273.703,Z 586.556,A -85,B 0,C 180,E1 -21280.754,E2 -21280.754} C_VEL
LIN {X 0,Y 268.25,Z 599.655,A -85,B 0,C 180,E1 -21281.694,E2 -21281.694} C_VEL
LIN {X 0,Y 261.118,Z 614.568,A -85,B 0,C 180,E1 -21283.105,E2 -21283.105} C_VEL
LIN {X 0,Y 254.288,Z 627.092,A -85,B 0,C 180,E1 -21284.626,E2 -21284.626} C_VEL
LIN {X 0,Y 246.06,Z 640.603,A -85,B 0,C 180,E1 -21286.723,E2 -21286.723} C_VEL
LIN {X 0,Y 238.438,Z 651.954,A -85,B 0,C 180,E1 -21289.015,E2 -21289.015} C_VEL
LIN {X 0,Y 231.371,Z 661.709,A -85,B 0,C 180,E1 -21291.484,E2 -21291.484} C_VEL
LIN {X 0,Y 224.82,Z 670.063,A -85,B 0,C 180,E1 -21294.114,E2 -21294.114} C_VEL
LIN {X 0,Y 218.903,Z 677.282,A -85,B 0,C 180,E1 -21296.918,E2 -21296.918} C_VEL
LIN {X 0,Y 213.158,Z 684.054,A -85,B 0,C 180,E1 -21300.356,E2 -21300.356} C_VEL
LIN {X 0,Y 208.251,Z 689.62,A -85,B 0,C 180,E1 -21303.975,E2 -21303.975} C_VEL
LIN {X 0,Y 204.076,Z 693.995,A -85,B 0,C 180,E1 -21307.737,E2 -21307.737} C_VEL
LIN {X 0,Y 200.985,Z 697.266,A -85,B 0,C 180,E1 -21311.654,E2 -21311.654} C_VEL
LIN {X 0,Y 198.904,Z 699.396,A -85,B 0,C 180,E1 -21315.677,E2 -21315.677} C_VEL
LIN {X 0,Y 197.728,Z 700.412,A -85,B 0,C 180,E1 -21319.76,E2 -21319.76} C_VEL
LIN {X 0,Y 197.25,Z 700.332,A -85,B 0,C 180,E1 -21323.861,E2 -21323.861} C_VEL
LIN {X 0,Y 197.361,Z 699.106,A -85,B 0,C 180,E1 -21327.956,E2 -21327.956} C_VEL
LIN {X 0,Y 197.523,Z 698.031,A -85,B 0,C 180,E1 -21329.997,E2 -21329.997} C_VEL
LIN {X 0,Y 197.536,Z 696.604,A -85,B 0,C 180,E1 -21332.036,E2 -21332.036} C_VEL
LIN {X 0,Y 197.489,Z 692.675,A -85,B 0,C 180,E1 -21336.125,E2 -21336.125} C_VEL
LIN {X 0,Y 197.785,Z 687.254,A -85,B 0,C 180,E1 -21340.231,E2 -21340.231} C_VEL
LIN {X 0,Y 198.69,Z 680.191,A -85,B 0,C 180,E1 -21344.332,E2 -21344.332} C_VEL
LIN {X 0,Y 200.051,Z 672.45,A -85,B 0,C 180,E1 -21347.899,E2 -21347.899} C_VEL
LIN {X 0,Y 201.999,Z 663.084,A -85,B 0,C 180,E1 -21351.424,E2 -21351.424} C_VEL
LIN {X 0,Y 204.622,Z 651.761,A -85,B 0,C 180,E1 -21354.878,E2 -21354.878} C_VEL
LIN {X 0,Y 207.299,Z 640.056,A -85,B 0,C 180,E1 -21357.782,E2 -21357.782} C_VEL
LIN {X 0,Y 209.986,Z 628.586,A -85,B 0,C 180,E1 -21360.131,E2 -21360.131} C_VEL
LIN {X 0,Y 212.929,Z 614.85,A -85,B 0,C 180,E1 -21362.432,E2 -21362.432} C_VEL
LIN {X 0,Y 215.96,Z 599.807,A -85,B 0,C 180,E1 -21364.429,E2 -21364.429} C_VEL
LIN {X 0,Y 218.609,Z 584.061,A -85,B 0,C 180,E1 -21366.063,E2 -21366.063} C_VEL
LIN {X 0,Y 220.89,Z 568.012,A -85,B 0,C 180,E1 -21367.306,E2 -21367.306} C_VEL
LIN {X 0,Y 222.598,Z 551.775,A -85,B 0,C 180,E1 -21368.197,E2 -21368.197} C_VEL
LIN {X 0,Y 229.86,Z 460.266,A -85,B 0,C 180,E1 -21372.023,E2 -21372.023} C_VEL
LIN {X 0,Y 221.357,Z 438.29,A -85,B 0,C 180,E1 -21374.389,E2 -21374.389} C_VEL
LIN {X 0,Y 211.935,Z 416.514,A -85,B 0,C 180,E1 -21377.152,E2 -21377.152} C_VEL
LIN {X 0,Y 203.433,Z 398.25,A -85,B 0,C 180,E1 -21379.79,E2 -21379.79} C_VEL
LIN {X 0,Y 200.944,Z 393.514,A -85,B 0,C 180,E1 -21380.58,E2 -21380.58} C_VEL
LIN {X 0,Y 199.746,Z 390.83,A -85,B 0,C 180,E1 -21380.994,E2 -21380.994} C_VEL
LIN {X 0,Y 199.631,Z 390.246,A -85,B 0,C 180,E1 -21381.122,E2 -21381.122} C_VEL
LIN {X 0,Y 199.599,Z 390.25,A -85,B 0,C 180,E1 -21385.711,E2 -21385.711} C_VEL
LIN {X 0,Y 199.674,Z 390.239,A -85,B 0,C 180,E1 -21388.133,E2 -21388.133} C_VEL
LIN {X 0,Y 199.622,Z 390.241,A -85,B 0,C 180,E1 -21392.763,E2 -21392.763} C_VEL
LIN {X 0,Y 199.658,Z 390.241,A -85,B 0,C 180,E1 -21397.22,E2 -21397.22} C_VEL
LIN {X 0,Y 199.733,Z 390.217,A -85,B 0,C 180,E1 -21401.802,E2 -21401.802} C_VEL
LIN {X 0,Y 199.781,Z 390.226,A -85,B 0,C 180,E1 -21405.745,E2 -21405.745} C_VEL
LIN {X 0,Y 200.01,Z 390.177,A -85,B 0,C 180,E1 -21409.882,E2 -21409.882} C_VEL
LIN {X 0,Y 199.986,Z 390.199,A -85,B 0,C 180,E1 -21413.949,E2 -21413.949} C_VEL
LIN {X 0,Y 200.272,Z 390.159,A -85,B 0,C 180,E1 -21417.99,E2 -21417.99} C_VEL
LIN {X 0,Y 200.434,Z 390.145,A -85,B 0,C 180,E1 -21420.001,E2 -21420.001} C_VEL
LIN {X 0,Y 199.975,Z 390.195,A -85,B 0,C 180,E1 -21424.031,E2 -21424.031} C_VEL
LIN {X 0,Y 200.062,Z 390.188,A -85,B 0,C 180,E1 -21428.078,E2 -21428.078} C_VEL
LIN {X 0,Y 199.841,Z 390.216,A -85,B 0,C 180,E1 -21432.182,E2 -21432.182} C_VEL
LIN {X 0,Y 199.732,Z 390.224,A -85,B 0,C 180,E1 -21436.35,E2 -21436.35} C_VEL
LIN {X 0,Y 199.633,Z 390.242,A -85,B 0,C 180,E1 -21440.613,E2 -21440.613} C_VEL
LIN {X 0,Y 199.615,Z 390.237,A -85,B 0,C 180,E1 -21444.993,E2 -21444.993} C_VEL
LIN {X 0,Y 199.597,Z 390.247,A -85,B 0,C 180,E1 -21449.536,E2 -21449.536} C_VEL
LIN {X 0,Y 199.655,Z 390.234,A -85,B 0,C 180,E1 -21452.355,E2 -21452.355} C_VEL
LIN {X 0,Y 199.608,Z 390.242,A -85,B 0,C 180,E1 -21456.767,E2 -21456.767} C_VEL
LIN {X 0,Y 199.586,Z 390.247,A -85,B 0,C 180,E1 -21459.334,E2 -21459.334} C_VEL
LIN {X 0,Y 199.559,Z 390.241,A -85,B 0,C 180,E1 -21462.31,E2 -21462.31} C_VEL
LIN {X 0,Y 199.568,Z 390.247,A -85,B 0,C 180,E1 -21465.23,E2 -21465.23} C_VEL
LIN {X 0,Y 199.562,Z 390.249,A -85,B 0,C 180,E1 -21468.005,E2 -21468.005} C_VEL
LIN {X 0,Y 199.59,Z 390.237,A -85,B 0,C 180,E1 -21470.776,E2 -21470.776} C_VEL
LIN {X 0,Y 199.606,Z 390.247,A -85,B 0,C 180,E1 -21475.716,E2 -21475.716} C_VEL
LIN {X 0,Y 199.681,Z 390.228,A -85,B 0,C 180,E1 -21478.137,E2 -21478.137} C_VEL
LIN {X 0,Y 199.632,Z 390.242,A -85,B 0,C 180,E1 -21482.767,E2 -21482.767} C_VEL
LIN {X 0,Y 199.677,Z 390.234,A -85,B 0,C 180,E1 -21487.225,E2 -21487.225} C_VEL
LIN {X 0,Y 199.749,Z 390.221,A -85,B 0,C 180,E1 -21491.802,E2 -21491.802} C_VEL
LIN {X 0,Y 199.819,Z 390.195,A -85,B 0,C 180,E1 -21495.75,E2 -21495.75} C_VEL
LIN {X 0,Y 200.024,Z 390.196,A -85,B 0,C 180,E1 -21499.885,E2 -21499.885} C_VEL
LIN {X 0,Y 200.003,Z 390.181,A -85,B 0,C 180,E1 -21503.952,E2 -21503.952} C_VEL
LIN {X 0,Y 200.29,Z 390.162,A -85,B 0,C 180,E1 -21507.992,E2 -21507.992} C_VEL
LIN {X 0,Y 200.451,Z 390.141,A -85,B 0,C 180,E1 -21510.003,E2 -21510.003} C_VEL
LIN {X 0,Y 199.995,Z 390.192,A -85,B 0,C 180,E1 -21514.033,E2 -21514.033} C_VEL
LIN {X 0,Y 200.079,Z 390.184,A -85,B 0,C 180,E1 -21518.08,E2 -21518.08} C_VEL
LIN {X 0,Y 199.863,Z 390.214,A -85,B 0,C 180,E1 -21522.183,E2 -21522.183} C_VEL
LIN {X 0,Y 199.756,Z 390.228,A -85,B 0,C 180,E1 -21526.35,E2 -21526.35} C_VEL
LIN {X 0,Y 199.681,Z 390.239,A -85,B 0,C 180,E1 -21530.745,E2 -21530.745} C_VEL
LIN {X 0,Y 200.753,Z 393.198,A -85,B 0,C 180,E1 -21531.166,E2 -21531.166} C_VEL
LIN {X 0,Y 202.359,Z 395.895,A -85,B 0,C 180,E1 -21531.658,E2 -21531.658} C_VEL
LIN {X 0,Y 212.388,Z 414.293,A -85,B 0,C 180,E1 -21534.587,E2 -21534.587} C_VEL
LIN {X 0,Y 223.019,Z 435.661,A -85,B 0,C 180,E1 -21537.489,E2 -21537.489} C_VEL
LIN {X 0,Y 227.413,Z 445.678,A -85,B 0,C 180,E1 -21538.653,E2 -21538.653} C_VEL
LIN {X 0,Y 229.798,Z 451.848,A -85,B 0,C 180,E1 -21539.299,E2 -21539.299} C_VEL
LIN {X 0,Y 222.144,Z 545.815,A -85,B 0,C 180,E1 -21543.236,E2 -21543.236} C_VEL
LIN {X 0,Y 220.297,Z 562.045,A -85,B 0,C 180,E1 -21544.275,E2 -21544.275} C_VEL
LIN {X 0,Y 218.13,Z 577.369,A -85,B 0,C 180,E1 -21545.617,E2 -21545.617} C_VEL
LIN {X 0,Y 215.475,Z 592.606,A -85,B 0,C 180,E1 -21547.342,E2 -21547.342} C_VEL
LIN {X 0,Y 212.59,Z 607.302,A -85,B 0,C 180,E1 -21549.451,E2 -21549.451} C_VEL
LIN {X 0,Y 209.614,Z 620.974,A -85,B 0,C 180,E1 -21551.89,E2 -21551.89} C_VEL
LIN {X 0,Y 206.904,Z 632.874,A -85,B 0,C 180,E1 -21554.494,E2 -21554.494} C_VEL
LIN {X 0,Y 204.458,Z 643.311,A -85,B 0,C 180,E1 -21557.243,E2 -21557.243} C_VEL
LIN {X 0,Y 202.234,Z 653.401,A -85,B 0,C 180,E1 -21560.446,E2 -21560.446} C_VEL
LIN {X 0,Y 200.377,Z 662.076,A -85,B 0,C 180,E1 -21563.779,E2 -21563.779} C_VEL
LIN {X 0,Y 198.908,Z 669.772,A -85,B 0,C 180,E1 -21567.395,E2 -21567.395} C_VEL
LIN {X 0,Y 197.888,Z 676.528,A -85,B 0,C 180,E1 -21571.35,E2 -21571.35} C_VEL
LIN {X 0,Y 197.285,Z 681.104,A -85,B 0,C 180,E1 -21574.691,E2 -21574.691} C_VEL
LIN {X 0,Y 196.901,Z 684.729,A -85,B 0,C 180,E1 -21578.135,E2 -21578.135} C_VEL
LIN {X 0,Y 196.805,Z 687.272,A -85,B 0,C 180,E1 -21581.252,E2 -21581.252} C_VEL
LIN {X 0,Y 197.144,Z 689.542,A -85,B 0,C 180,E1 -21585.549,E2 -21585.549} C_VEL
LIN {X 0,Y 197.977,Z 690.5,A -85,B 0,C 180,E1 -21589.776,E2 -21589.776} C_VEL
LIN {X 0,Y 199.58,Z 690.253,A -85,B 0,C 180,E1 -21593.935,E2 -21593.935} C_VEL
LIN {X 0,Y 201.913,Z 688.876,A -85,B 0,C 180,E1 -21598.005,E2 -21598.005} C_VEL
LIN {X 0,Y 205.114,Z 686.353,A -85,B 0,C 180,E1 -21601.963,E2 -21601.963} C_VEL
LIN {X 0,Y 209.26,Z 682.673,A -85,B 0,C 180,E1 -21605.782,E2 -21605.782} C_VEL
LIN {X 0,Y 214.233,Z 677.719,A -85,B 0,C 180,E1 -21609.44,E2 -21609.44} C_VEL
LIN {X 0,Y 220.148,Z 671.474,A -85,B 0,C 180,E1 -21612.912,E2 -21612.912} C_VEL
LIN {X 0,Y 226.933,Z 663.707,A -85,B 0,C 180,E1 -21616.184,E2 -21616.184} C_VEL
LIN {X 0,Y 233.515,Z 655.603,A -85,B 0,C 180,E1 -21618.877,E2 -21618.877} C_VEL
LIN {X 0,Y 241.887,Z 644.331,A -85,B 0,C 180,E1 -21621.788,E2 -21621.788} C_VEL
LIN {X 0,Y 249.574,Z 632.826,A -85,B 0,C 180,E1 -21624.099,E2 -21624.099} C_VEL
LIN {X 0,Y 257.457,Z 619.648,A -85,B 0,C 180,E1 -21626.148,E2 -21626.148} C_VEL
LIN {X 0,Y 264.014,Z 607.177,A -85,B 0,C 180,E1 -21627.697,E2 -21627.697} C_VEL
LIN {X 0,Y 270.092,Z 594.074,A -85,B 0,C 180,E1 -21628.988,E2 -21628.988} C_VEL
LIN {X 0,Y 275.737,Z 579.864,A -85,B 0,C 180,E1 -21630.072,E2 -21630.072} C_VEL
LIN {X 0,Y 280.609,Z 564.875,A -85,B 0,C 180,E1 -21630.941,E2 -21630.941} C_VEL
LIN {X 0,Y 284.589,Z 549.649,A -85,B 0,C 180,E1 -21631.601,E2 -21631.601} C_VEL
LIN {X 0,Y 294.204,Z 501.868,A -85,B 0,C 180,E1 -21633.194,E2 -21633.194} C_VEL
LIN {X 0,Y 294.303,Z 501.141,A -85,B 0,C 180,E1 -21633.382,E2 -21633.382} C_VEL
LIN {X 0,Y 294.082,Z 501.563,A -85,B 0,C 180,E1 -21633.898,E2 -21633.898} C_VEL
LIN {X 0,Y 292.967,Z 505.838,A -85,B 0,C 180,E1 -21635.313,E2 -21635.313} C_VEL
LIN {X 0,Y 292.881,Z 506.397,A -85,B 0,C 180,E1 -21635.737,E2 -21635.737} C_VEL
LIN {X 0,Y 292.886,Z 506.73,A -85,B 0,C 180,E1 -21636.178,E2 -21636.178} C_VEL
LIN {X 0,Y 282.589,Z 555.17,A -85,B 0,C 180,E1 -21637.774,E2 -21637.774} C_VEL
LIN {X 0,Y 278.063,Z 570.884,A -85,B 0,C 180,E1 -21638.413,E2 -21638.413} C_VEL
LIN {X 0,Y 272.328,Z 586.607,A -85,B 0,C 180,E1 -21639.264,E2 -21639.264} C_VEL
LIN {X 0,Y 266.025,Z 601.026,A -85,B 0,C 180,E1 -21640.282,E2 -21640.282} C_VEL
LIN {X 0,Y 259.299,Z 614.346,A -85,B 0,C 180,E1 -21641.516,E2 -21641.516} C_VEL
LIN {X 0,Y 251.535,Z 627.782,A -85,B 0,C 180,E1 -21643.116,E2 -21643.116} C_VEL
LIN {X 0,Y 243.585,Z 640.154,A -85,B 0,C 180,E1 -21645.015,E2 -21645.015} C_VEL
LIN {X 0,Y 234.475,Z 652.958,A -85,B 0,C 180,E1 -21647.589,E2 -21647.589} C_VEL
LIN {X 0,Y 227.046,Z 662.406,A -85,B 0,C 180,E1 -21650.034,E2 -21650.034} C_VEL
LIN {X 0,Y 219.184,Z 671.754,A -85,B 0,C 180,E1 -21653.098,E2 -21653.098} C_VEL
LIN {X 0,Y 211.5,Z 680.226,A -85,B 0,C 180,E1 -21656.748,E2 -21656.748} C_VEL
LIN {X 0,Y 205.671,Z 686.41,A -85,B 0,C 180,E1 -21660.296,E2 -21660.296} C_VEL
LIN {X 0,Y 200.731,Z 691.397,A -85,B 0,C 180,E1 -21664.043,E2 -21664.043} C_VEL
LIN {X 0,Y 197.523,Z 694.415,A -85,B 0,C 180,E1 -21666.956,E2 -21666.956} C_VEL
LIN {X 0,Y 194.215,Z 697.42,A -85,B 0,C 180,E1 -21670.99,E2 -21670.99} C_VEL
LIN {X 0,Y 191.997,Z 699.377,A -85,B 0,C 180,E1 -21675.15,E2 -21675.15} C_VEL
LIN {X 0,Y 190.706,Z 700.241,A -85,B 0,C 180,E1 -21679.379,E2 -21679.379} C_VEL
LIN {X 0,Y 190.177,Z 699.959,A -85,B 0,C 180,E1 -21683.632,E2 -21683.632} C_VEL
LIN {X 0,Y 190.305,Z 698.553,A -85,B 0,C 180,E1 -21687.88,E2 -21687.88} C_VEL
LIN {X 0,Y 190.46,Z 697.4,A -85,B 0,C 180,E1 -21689.997,E2 -21689.997} C_VEL
LIN {X 0,Y 190.474,Z 695.891,A -85,B 0,C 180,E1 -21692.111,E2 -21692.111} C_VEL
LIN {X 0,Y 190.429,Z 691.788,A -85,B 0,C 180,E1 -21696.353,E2 -21696.353} C_VEL
LIN {X 0,Y 190.775,Z 686.151,A -85,B 0,C 180,E1 -21700.611,E2 -21700.611} C_VEL
LIN {X 0,Y 191.777,Z 678.834,A -85,B 0,C 180,E1 -21704.861,E2 -21704.861} C_VEL
LIN {X 0,Y 193.24,Z 670.903,A -85,B 0,C 180,E1 -21708.552,E2 -21708.552} C_VEL
LIN {X 0,Y 195.328,Z 661.279,A -85,B 0,C 180,E1 -21712.194,E2 -21712.194} C_VEL
LIN {X 0,Y 197.653,Z 651.465,A -85,B 0,C 180,E1 -21715.254,E2 -21715.254} C_VEL
LIN {X 0,Y 200.421,Z 639.75,A -85,B 0,C 180,E1 -21718.251,E2 -21718.251} C_VEL
LIN {X 0,Y 203.423,Z 627.08,A -85,B 0,C 180,E1 -21720.892,E2 -21720.892} C_VEL
LIN {X 0,Y 206.206,Z 614.486,A -85,B 0,C 180,E1 -21723.042,E2 -21723.042} C_VEL
LIN {X 0,Y 208.942,Z 601.298,A -85,B 0,C 180,E1 -21724.873,E2 -21724.873} C_VEL
LIN {X 0,Y 211.671,Z 586.02,A -85,B 0,C 180,E1 -21726.549,E2 -21726.549} C_VEL
LIN {X 0,Y 214.057,Z 570.128,A -85,B 0,C 180,E1 -21727.865,E2 -21727.865} C_VEL
LIN {X 0,Y 215.865,Z 554.362,A -85,B 0,C 180,E1 -21728.805,E2 -21728.805} C_VEL
LIN {X 0,Y 223.434,Z 461.839,A -85,B 0,C 180,E1 -21732.808,E2 -21732.808} C_VEL
LIN {X 0,Y 214.757,Z 439.358,A -85,B 0,C 180,E1 -21735.356,E2 -21735.356} C_VEL
LIN {X 0,Y 205.126,Z 417.158,A -85,B 0,C 180,E1 -21738.283,E2 -21738.283} C_VEL
LIN {X 0,Y 197.769,Z 401.385,A -85,B 0,C 180,E1 -21740.701,E2 -21740.701} C_VEL
LIN {X 0,Y 194.302,Z 394.935,A -85,B 0,C 180,E1 -21741.832,E2 -21741.832} C_VEL
LIN {X 0,Y 192.824,Z 392.297,A -85,B 0,C 180,E1 -21742.322,E2 -21742.322} C_VEL
LIN {X 0,Y 192.576,Z 391.127,A -85,B 0,C 180,E1 -21742.507,E2 -21742.507} C_VEL
LIN {X 0,Y 192.594,Z 391.122,A -85,B 0,C 180,E1 -21747.06,E2 -21747.06} C_VEL
LIN {X 0,Y 192.607,Z 391.119,A -85,B 0,C 180,E1 -21751.683,E2 -21751.683} C_VEL
LIN {X 0,Y 192.645,Z 391.112,A -85,B 0,C 180,E1 -21756.341,E2 -21756.341} C_VEL
LIN {X 0,Y 192.682,Z 391.094,A -85,B 0,C 180,E1 -21761.491,E2 -21761.491} C_VEL
LIN {X 0,Y 192.708,Z 391.106,A -85,B 0,C 180,E1 -21765.21,E2 -21765.21} C_VEL
LIN {X 0,Y 192.933,Z 391.057,A -85,B 0,C 180,E1 -21769.567,E2 -21769.567} C_VEL
LIN {X 0,Y 192.951,Z 391.074,A -85,B 0,C 180,E1 -21773.727,E2 -21773.727} C_VEL
LIN {X 0,Y 193.217,Z 391.037,A -85,B 0,C 180,E1 -21777.916,E2 -21777.916} C_VEL
LIN {X 0,Y 193.401,Z 391.021,A -85,B 0,C 180,E1 -21780.001,E2 -21780.001} C_VEL
LIN {X 0,Y 192.922,Z 391.074,A -85,B 0,C 180,E1 -21784.179,E2 -21784.179} C_VEL
LIN {X 0,Y 193.013,Z 391.064,A -85,B 0,C 180,E1 -21788.375,E2 -21788.375} C_VEL
LIN {X 0,Y 192.768,Z 391.097,A -85,B 0,C 180,E1 -21792.636,E2 -21792.636} C_VEL
LIN {X 0,Y 192.693,Z 391.099,A -85,B 0,C 180,E1 -21796.965,E2 -21796.965} C_VEL
LIN {X 0,Y 192.567,Z 391.122,A -85,B 0,C 180,E1 -21801.406,E2 -21801.406} C_VEL
LIN {X 0,Y 192.61,Z 391.111,A -85,B 0,C 180,E1 -21804.197,E2 -21804.197} C_VEL
LIN {X 0,Y 192.59,Z 391.118,A -85,B 0,C 180,E1 -21808.867,E2 -21808.867} C_VEL
LIN {X 0,Y 192.585,Z 391.113,A -85,B 0,C 180,E1 -21813.189,E2 -21813.189} C_VEL
LIN {X 0,Y 192.533,Z 391.126,A -85,B 0,C 180,E1 -21818.357,E2 -21818.357} C_VEL
LIN {X 0,Y 192.478,Z 391.123,A -85,B 0,C 180,E1 -21823.097,E2 -21823.097} C_VEL
LIN {X 0,Y 192.477,Z 391.132,A -85,B 0,C 180,E1 -21826.91,E2 -21826.91} C_VEL
LIN {X 0,Y 192.535,Z 391.118,A -85,B 0,C 180,E1 -21831.649,E2 -21831.649} C_VEL
LIN {X 0,Y 192.59,Z 391.116,A -85,B 0,C 180,E1 -21836.817,E2 -21836.817} C_VEL
LIN {X 0,Y 192.615,Z 391.118,A -85,B 0,C 180,E1 -21841.688,E2 -21841.688} C_VEL
LIN {X 0,Y 192.664,Z 391.107,A -85,B 0,C 180,E1 -21846.347,E2 -21846.347} C_VEL
LIN {X 0,Y 192.698,Z 391.101,A -85,B 0,C 180,E1 -21851.491,E2 -21851.491} C_VEL
LIN {X 0,Y 192.743,Z 391.072,A -85,B 0,C 180,E1 -21855.216,E2 -21855.216} C_VEL
LIN {X 0,Y 192.946,Z 391.075,A -85,B 0,C 180,E1 -21859.57,E2 -21859.57} C_VEL
LIN {X 0,Y 192.967,Z 391.058,A -85,B 0,C 180,E1 -21863.73,E2 -21863.73} C_VEL
LIN {X 0,Y 193.234,Z 391.04,A -85,B 0,C 180,E1 -21867.919,E2 -21867.919} C_VEL
LIN {X 0,Y 193.417,Z 391.018,A -85,B 0,C 180,E1 -21870.003,E2 -21870.003} C_VEL
LIN {X 0,Y 192.943,Z 391.071,A -85,B 0,C 180,E1 -21874.181,E2 -21874.181} C_VEL
LIN {X 0,Y 193.03,Z 391.06,A -85,B 0,C 180,E1 -21878.377,E2 -21878.377} C_VEL
LIN {X 0,Y 192.784,Z 391.095,A -85,B 0,C 180,E1 -21882.638,E2 -21882.638} C_VEL
LIN {X 0,Y 192.702,Z 391.1,A -85,B 0,C 180,E1 -21888.512,E2 -21888.512} C_VEL
LIN {X 0,Y 192.638,Z 391.112,A -85,B 0,C 180,E1 -21889.379,E2 -21889.379} C_VEL
LIN {X 0,Y 193.687,Z 394.058,A -85,B 0,C 180,E1 -21889.804,E2 -21889.804} C_VEL
LIN {X 0,Y 195.096,Z 396.412,A -85,B 0,C 180,E1 -21890.251,E2 -21890.251} C_VEL
LIN {X 0,Y 203.845,Z 412.112,A -85,B 0,C 180,E1 -21892.963,E2 -21892.963} C_VEL
LIN {X 0,Y 215.22,Z 434.569,A -85,B 0,C 180,E1 -21896.222,E2 -21896.222} C_VEL
LIN {X 0,Y 220.603,Z 446.479,A -85,B 0,C 180,E1 -21897.723,E2 -21897.723} C_VEL
LIN {X 0,Y 223.356,Z 453.757,A -85,B 0,C 180,E1 -21898.518,E2 -21898.518} C_VEL
LIN {X 0,Y 215.654,Z 545.98,A -85,B 0,C 180,E1 -21902.498,E2 -21902.498} C_VEL
LIN {X 0,Y 213.885,Z 561.001,A -85,B 0,C 180,E1 -21903.464,E2 -21903.464} C_VEL
LIN {X 0,Y 211.563,Z 577.186,A -85,B 0,C 180,E1 -21904.904,E2 -21904.904} C_VEL
LIN {X 0,Y 208.801,Z 592.655,A -85,B 0,C 180,E1 -21906.696,E2 -21906.696} C_VEL
LIN {X 0,Y 206.029,Z 606.435,A -85,B 0,C 180,E1 -21908.711,E2 -21908.711} C_VEL
LIN {X 0,Y 202.898,Z 620.522,A -85,B 0,C 180,E1 -21911.267,E2 -21911.267} C_VEL
LIN {X 0,Y 200.012,Z 632.816,A -85,B 0,C 180,E1 -21914.03,E2 -21914.03} C_VEL
LIN {X 0,Y 197.556,Z 642.957,A -85,B 0,C 180,E1 -21916.778,E2 -21916.778} C_VEL
LIN {X 0,Y 195.133,Z 653.583,A -85,B 0,C 180,E1 -21920.26,E2 -21920.26} C_VEL
LIN {X 0,Y 193.265,Z 662.188,A -85,B 0,C 180,E1 -21923.691,E2 -21923.691} C_VEL
LIN {X 0,Y 191.798,Z 669.911,A -85,B 0,C 180,E1 -21927.44,E2 -21927.44} C_VEL
LIN {X 0,Y 190.78,Z 676.471,A -85,B 0,C 180,E1 -21931.386,E2 -21931.386} C_VEL
LIN {X 0,Y 190.168,Z 681.097,A -85,B 0,C 180,E1 -21934.848,E2 -21934.848} C_VEL
LIN {X 0,Y 189.816,Z 684.637,A -85,B 0,C 180,E1 -21938.268,E2 -21938.268} C_VEL
LIN {X 0,Y 189.781,Z 688.021,A -85,B 0,C 180,E1 -21942.766,E2 -21942.766} C_VEL
LIN {X 0,Y 190.273,Z 690.039,A -85,B 0,C 180,E1 -21947.195,E2 -21947.195} C_VEL
LIN {X 0,Y 191.63,Z 690.804,A -85,B 0,C 180,E1 -21951.997,E2 -21951.997} C_VEL
LIN {X 0,Y 193.364,Z 690.397,A -85,B 0,C 180,E1 -21955.831,E2 -21955.831} C_VEL
LIN {X 0,Y 196.811,Z 688.409,A -85,B 0,C 180,E1 -21960.789,E2 -21960.789} C_VEL
LIN {X 0,Y 199.889,Z 686.115,A -85,B 0,C 180,E1 -21964.032,E2 -21964.032} C_VEL
LIN {X 0,Y 204.554,Z 682.241,A -85,B 0,C 180,E1 -21967.899,E2 -21967.899} C_VEL
LIN {X 0,Y 210.14,Z 677.191,A -85,B 0,C 180,E1 -21971.575,E2 -21971.575} C_VEL
LIN {X 0,Y 216.636,Z 670.771,A -85,B 0,C 180,E1 -21975.042,E2 -21975.042} C_VEL
LIN {X 0,Y 224,Z 662.878,A -85,B 0,C 180,E1 -21978.285,E2 -21978.285} C_VEL
LIN {X 0,Y 232.181,Z 653.262,A -85,B 0,C 180,E1 -21981.298,E2 -21981.298} C_VEL
LIN {X 0,Y 239.596,Z 643.702,A -85,B 0,C 180,E1 -21983.635,E2 -21983.635} C_VEL
LIN {X 0,Y 247.052,Z 633.146,A -85,B 0,C 180,E1 -21985.71,E2 -21985.71} C_VEL
LIN {X 0,Y 255.104,Z 620.269,A -85,B 0,C 180,E1 -21987.694,E2 -21987.694} C_VEL
LIN {X 0,Y 262.335,Z 607.333,A -85,B 0,C 180,E1 -21989.269,E2 -21989.269} C_VEL
LIN {X 0,Y 268.507,Z 594.592,A -85,B 0,C 180,E1 -21990.473,E2 -21990.473} C_VEL
LIN {X 0,Y 274.704,Z 579.648,A -85,B 0,C 180,E1 -21991.592,E2 -21991.592} C_VEL
LIN {X 0,Y 279.643,Z 565.214,A -85,B 0,C 180,E1 -21992.386,E2 -21992.386} C_VEL
LIN {X 0,Y 283.506,Z 550.946,A -85,B 0,C 180,E1 -21992.997,E2 -21992.997} C_VEL
LIN {X 0,Y 292.996,Z 506.07,A -85,B 0,C 180,E1 -21994.471,E2 -21994.471} C_VEL
LIN {X 0,Y 292.881,Z 506.397,A -85,B 0,C 180,E1 -21995.737,E2 -21995.737} C_VEL
LIN {X 0,Y 292.756,Z 507.23,A -85,B 0,C 180,E1 -21996.064,E2 -21996.064} C_VEL
LIN {X 0,Y 292.236,Z 509.925,A -85,B 0,C 180,E1 -21996.382,E2 -21996.382} C_VEL
LIN {X 0,Y 291.599,Z 512.958,A -85,B 0,C 180,E1 -21996.478,E2 -21996.478} C_VEL
LIN {X 0,Y 290.784,Z 516.682,A -85,B 0,C 180,E1 -21996.443,E2 -21996.443} C_VEL
LIN {X 0,Y 287.705,Z 530.297,A -85,B 0,C 180,E1 -21995.759,E2 -21995.759} C_VEL
LIN {X 0,Y 286.66,Z 535.065,A -85,B 0,C 180,E1 -21995.689,E2 -21995.689} C_VEL
LIN {X 0,Y 286.155,Z 537.436,A -85,B 0,C 180,E1 -21995.744,E2 -21995.744} C_VEL
LIN {X 0,Y 281.569,Z 557.158,A -85,B 0,C 180,E1 -21996.391,E2 -21996.391} C_VEL
LIN {X 0,Y 276.726,Z 572.689,A -85,B 0,C 180,E1 -21997.018,E2 -21997.018} C_VEL
LIN {X 0,Y 270.489,Z 588.778,A -85,B 0,C 180,E1 -21997.884,E2 -21997.884} C_VEL
LIN {X 0,Y 264.005,Z 602.705,A -85,B 0,C 180,E1 -21998.86,E2 -21998.86} C_VEL
LIN {X 0,Y 256.372,Z 616.732,A -85,B 0,C 180,E1 -22000.166,E2 -22000.166} C_VEL
LIN {X 0,Y 249.034,Z 628.712,A -85,B 0,C 180,E1 -22001.592,E2 -22001.592} C_VEL
LIN {X 0,Y 240.148,Z 641.612,A -85,B 0,C 180,E1 -22003.585,E2 -22003.585} C_VEL
LIN {X 0,Y 231.82,Z 652.588,A -85,B 0,C 180,E1 -22005.788,E2 -22005.788} C_VEL
LIN {X 0,Y 222.917,Z 663.248,A -85,B 0,C 180,E1 -22008.539,E2 -22008.539} C_VEL
LIN {X 0,Y 214.728,Z 672.202,A -85,B 0,C 180,E1 -22011.544,E2 -22011.544} C_VEL
LIN {X 0,Y 207.341,Z 679.73,A -85,B 0,C 180,E1 -22014.811,E2 -22014.811} C_VEL
LIN {X 0,Y 201.023,Z 685.878,A -85,B 0,C 180,E1 -22018.368,E2 -22018.368} C_VEL
LIN {X 0,Y 195.594,Z 690.9,A -85,B 0,C 180,E1 -22022.15,E2 -22022.15} C_VEL
LIN {X 0,Y 190.989,Z 694.819,A -85,B 0,C 180,E1 -22026.12,E2 -22026.12} C_VEL
LIN {X 0,Y 187.476,Z 697.604,A -85,B 0,C 180,E1 -22030.279,E2 -22030.279} C_VEL
LIN {X 0,Y 185.108,Z 699.317,A -85,B 0,C 180,E1 -22034.584,E2 -22034.584} C_VEL
LIN {X 0,Y 183.701,Z 700.002,A -85,B 0,C 180,E1 -22038.969,E2 -22038.969} C_VEL
LIN {X 0,Y 183.097,Z 699.587,A -85,B 0,C 180,E1 -22043.384,E2 -22043.384} C_VEL
LIN {X 0,Y 183.25,Z 697.98,A -85,B 0,C 180,E1 -22047.799,E2 -22047.799} C_VEL
LIN {X 0,Y 183.398,Z 696.724,A -85,B 0,C 180,E1 -22049.997,E2 -22049.997} C_VEL
LIN {X 0,Y 183.413,Z 695.126,A -85,B 0,C 180,E1 -22052.193,E2 -22052.193} C_VEL
LIN {X 0,Y 183.377,Z 692.746,A -85,B 0,C 180,E1 -22054.827,E2 -22054.827} C_VEL
LIN {X 0,Y 183.484,Z 688.118,A -85,B 0,C 180,E1 -22058.81,E2 -22058.81} C_VEL
LIN {X 0,Y 184.204,Z 681.427,A -85,B 0,C 180,E1 -22063.23,E2 -22063.23} C_VEL
LIN {X 0,Y 185.417,Z 674.1,A -85,B 0,C 180,E1 -22067.079,E2 -22067.079} C_VEL
LIN {X 0,Y 187.318,Z 665.207,A -85,B 0,C 180,E1 -22070.878,E2 -22070.878} C_VEL
LIN {X 0,Y 189.897,Z 654.446,A -85,B 0,C 180,E1 -22074.601,E2 -22074.601} C_VEL
LIN {X 0,Y 192.762,Z 642.35,A -85,B 0,C 180,E1 -22077.992,E2 -22077.992} C_VEL
LIN {X 0,Y 195.817,Z 630.181,A -85,B 0,C 180,E1 -22080.756,E2 -22080.756} C_VEL
LIN {X 0,Y 198.861,Z 616.931,A -85,B 0,C 180,E1 -22083.211,E2 -22083.211} C_VEL
LIN {X 0,Y 201.967,Z 602.578,A -85,B 0,C 180,E1 -22085.342,E2 -22085.342} C_VEL
LIN {X 0,Y 204.784,Z 587.873,A -85,B 0,C 180,E1 -22087.061,E2 -22087.061} C_VEL
LIN {X 0,Y 207.177,Z 572.825,A -85,B 0,C 180,E1 -22088.413,E2 -22088.413} C_VEL
LIN {X 0,Y 209.167,Z 556.519,A -85,B 0,C 180,E1 -22089.477,E2 -22089.477} C_VEL
LIN {X 0,Y 217.092,Z 463.713,A -85,B 0,C 180,E1 -22093.613,E2 -22093.613} C_VEL
LIN {X 0,Y 209.149,Z 442.913,A -85,B 0,C 180,E1 -22096.044,E2 -22096.044} C_VEL
LIN {X 0,Y 199.85,Z 421.167,A -85,B 0,C 180,E1 -22099,E2 -22099} C_VEL
LIN {X 0,Y 192.246,Z 404.82,A -85,B 0,C 180,E1 -22101.577,E2 -22101.577} C_VEL
LIN {X 0,Y 187.015,Z 395.541,A -85,B 0,C 180,E1 -22103.348,E2 -22103.348} C_VEL
LIN {X 0,Y 185.701,Z 392.971,A -85,B 0,C 180,E1 -22103.832,E2 -22103.832} C_VEL
LIN {X 0,Y 185.533,Z 392.005,A -85,B 0,C 180,E1 -22103.963,E2 -22103.963} C_VEL
LIN {X 0,Y 185.519,Z 392.002,A -85,B 0,C 180,E1 -22107.971,E2 -22107.971} C_VEL
LIN {X 0,Y 185.535,Z 391.998,A -85,B 0,C 180,E1 -22110.594,E2 -22110.594} C_VEL
LIN {X 0,Y 185.532,Z 391.992,A -85,B 0,C 180,E1 -22115.375,E2 -22115.375} C_VEL
LIN {X 0,Y 185.613,Z 391.973,A -85,B 0,C 180,E1 -22121.178,E2 -22121.178} C_VEL
LIN {X 0,Y 185.693,Z 391.975,A -85,B 0,C 180,E1 -22126.875,E2 -22126.875} C_VEL
LIN {X 0,Y 185.959,Z 391.935,A -85,B 0,C 180,E1 -22131.306,E2 -22131.306} C_VEL
LIN {X 0,Y 186.163,Z 391.915,A -85,B 0,C 180,E1 -22137.837,E2 -22137.837} C_VEL
LIN {X 0,Y 186.367,Z 391.897,A -85,B 0,C 180,E1 -22140.001,E2 -22140.001} C_VEL
LIN {X 0,Y 185.87,Z 391.953,A -85,B 0,C 180,E1 -22144.338,E2 -22144.338} C_VEL
LIN {X 0,Y 185.962,Z 391.941,A -85,B 0,C 180,E1 -22148.695,E2 -22148.695} C_VEL
LIN {X 0,Y 185.693,Z 391.978,A -85,B 0,C 180,E1 -22153.126,E2 -22153.126} C_VEL
LIN {X 0,Y 185.614,Z 391.983,A -85,B 0,C 180,E1 -22158.823,E2 -22158.823} C_VEL
LIN {X 0,Y 185.534,Z 391.99,A -85,B 0,C 180,E1 -22164.626,E2 -22164.626} C_VEL
LIN {X 0,Y 185.534,Z 391.998,A -85,B 0,C 180,E1 -22169.502,E2 -22169.502} C_VEL
LIN {X 0,Y 185.488,Z 391.994,A -85,B 0,C 180,E1 -22174.635,E2 -22174.635} C_VEL
LIN {X 0,Y 185.491,Z 392.001,A -85,B 0,C 180,E1 -22177.317,E2 -22177.317} C_VEL
LIN {X 0,Y 185.454,Z 392.003,A -85,B 0,C 180,E1 -22180.724,E2 -22180.724} C_VEL
LIN {X 0,Y 185.448,Z 392.01,A -85,B 0,C 180,E1 -22186.06,E2 -22186.06} C_VEL
LIN {X 0,Y 185.449,Z 392,A -85,B 0,C 180,E1 -22189.895,E2 -22189.895} C_VEL
LIN {X 0,Y 185.495,Z 392,A -85,B 0,C 180,E1 -22192.717,E2 -22192.717} C_VEL
LIN {X 0,Y 185.526,Z 391.991,A -85,B 0,C 180,E1 -22197.976,E2 -22197.976} C_VEL
LIN {X 0,Y 185.543,Z 391.996,A -85,B 0,C 180,E1 -22200.599,E2 -22200.599} C_VEL
LIN {X 0,Y 185.56,Z 391.989,A -85,B 0,C 180,E1 -22205.382,E2 -22205.382} C_VEL
LIN {X 0,Y 185.632,Z 391.983,A -85,B 0,C 180,E1 -22211.175,E2 -22211.175} C_VEL
LIN {X 0,Y 185.672,Z 391.952,A -85,B 0,C 180,E1 -22214.639,E2 -22214.639} C_VEL
LIN {X 0,Y 185.889,Z 391.953,A -85,B 0,C 180,E1 -22219.423,E2 -22219.423} C_VEL
LIN {X 0,Y 185.932,Z 391.935,A -85,B 0,C 180,E1 -22223.492,E2 -22223.492} C_VEL
LIN {X 0,Y 186.179,Z 391.917,A -85,B 0,C 180,E1 -22227.84,E2 -22227.84} C_VEL
LIN {X 0,Y 186.383,Z 391.894,A -85,B 0,C 180,E1 -22230.003,E2 -22230.003} C_VEL
LIN {X 0,Y 185.891,Z 391.951,A -85,B 0,C 180,E1 -22234.34,E2 -22234.34} C_VEL
LIN {X 0,Y 185.979,Z 391.936,A -85,B 0,C 180,E1 -22238.697,E2 -22238.697} C_VEL
LIN {X 0,Y 185.707,Z 391.973,A -85,B 0,C 180,E1 -22243.128,E2 -22243.128} C_VEL
LIN {X 0,Y 185.665,Z 392.026,A -85,B 0,C 180,E1 -22247.917,E2 -22247.917} C_VEL
LIN {X 0,Y 186.625,Z 394.781,A -85,B 0,C 180,E1 -22248.337,E2 -22248.337} C_VEL
LIN {X 0,Y 187.937,Z 396.938,A -85,B 0,C 180,E1 -22248.784,E2 -22248.784} C_VEL
LIN {X 0,Y 197.549,Z 414.203,A -85,B 0,C 180,E1 -22251.903,E2 -22251.903} C_VEL
LIN {X 0,Y 207.466,Z 433.827,A -85,B 0,C 180,E1 -22254.93,E2 -22254.93} C_VEL
LIN {X 0,Y 214.603,Z 449.02,A -85,B 0,C 180,E1 -22256.952,E2 -22256.952} C_VEL
LIN {X 0,Y 217.042,Z 455.439,A -85,B 0,C 180,E1 -22257.689,E2 -22257.689} C_VEL
LIN {X 0,Y 209.149,Z 546.313,A -85,B 0,C 180,E1 -22261.725,E2 -22261.725} C_VEL
LIN {X 0,Y 207.183,Z 562.371,A -85,B 0,C 180,E1 -22262.816,E2 -22262.816} C_VEL
LIN {X 0,Y 204.966,Z 577.249,A -85,B 0,C 180,E1 -22264.192,E2 -22264.192} C_VEL
LIN {X 0,Y 202.093,Z 592.81,A -85,B 0,C 180,E1 -22266.052,E2 -22266.052} C_VEL
LIN {X 0,Y 199.092,Z 607.213,A -85,B 0,C 180,E1 -22268.238,E2 -22268.238} C_VEL
LIN {X 0,Y 196.155,Z 620.067,A -85,B 0,C 180,E1 -22270.652,E2 -22270.652} C_VEL
LIN {X 0,Y 193.318,Z 631.889,A -85,B 0,C 180,E1 -22273.356,E2 -22273.356} C_VEL
LIN {X 0,Y 190.678,Z 642.493,A -85,B 0,C 180,E1 -22276.276,E2 -22276.276} C_VEL
LIN {X 0,Y 188.158,Z 653.253,A -85,B 0,C 180,E1 -22279.885,E2 -22279.885} C_VEL
LIN {X 0,Y 186.198,Z 662.142,A -85,B 0,C 180,E1 -22283.524,E2 -22283.524} C_VEL
LIN {X 0,Y 184.594,Z 670.591,A -85,B 0,C 180,E1 -22287.79,E2 -22287.79} C_VEL
LIN {X 0,Y 183.615,Z 676.763,A -85,B 0,C 180,E1 -22291.689,E2 -22291.689} C_VEL
LIN {X 0,Y 183.042,Z 681.025,A -85,B 0,C 180,E1 -22295.016,E2 -22295.016} C_VEL
LIN {X 0,Y 182.686,Z 684.628,A -85,B 0,C 180,E1 -22298.563,E2 -22298.563} C_VEL
LIN {X 0,Y 182.621,Z 687.381,A -85,B 0,C 180,E1 -22302.068,E2 -22302.068} C_VEL
LIN {X 0,Y 182.839,Z 688.762,A -85,B 0,C 180,E1 -22304.391,E2 -22304.391} C_VEL
LIN {X 0,Y 183.513,Z 690.51,A -85,B 0,C 180,E1 -22308.96,E2 -22308.96} C_VEL
LIN {X 0,Y 185.067,Z 691.06,A -85,B 0,C 180,E1 -22313.458,E2 -22313.458} C_VEL
LIN {X 0,Y 187.404,Z 690.475,A -85,B 0,C 180,E1 -22317.85,E2 -22317.85} C_VEL
LIN {X 0,Y 190.705,Z 688.778,A -85,B 0,C 180,E1 -22322.111,E2 -22322.111} C_VEL
LIN {X 0,Y 194.987,Z 685.897,A -85,B 0,C 180,E1 -22326.207,E2 -22326.207} C_VEL
LIN {X 0,Y 200.205,Z 681.893,A -85,B 0,C 180,E1 -22330.108,E2 -22330.108} C_VEL
LIN {X 0,Y 206.393,Z 676.661,A -85,B 0,C 180,E1 -22333.789,E2 -22333.789} C_VEL
LIN {X 0,Y 213.531,Z 670.083,A -85,B 0,C 180,E1 -22337.23,E2 -22337.23} C_VEL
LIN {X 0,Y 221.439,Z 662.068,A -85,B 0,C 180,E1 -22340.433,E2 -22340.433} C_VEL
LIN {X 0,Y 229.127,Z 653.531,A -85,B 0,C 180,E1 -22343.041,E2 -22343.041} C_VEL
LIN {X 0,Y 237.336,Z 643.618,A -85,B 0,C 180,E1 -22345.427,E2 -22345.427} C_VEL
LIN {X 0,Y 244.746,Z 633.599,A -85,B 0,C 180,E1 -22347.351,E2 -22347.351} C_VEL
LIN {X 0,Y 252.554,Z 621.958,A -85,B 0,C 180,E1 -22349.142,E2 -22349.142} C_VEL
LIN {X 0,Y 260.735,Z 608.021,A -85,B 0,C 180,E1 -22350.806,E2 -22350.806} C_VEL
LIN {X 0,Y 267.741,Z 594.257,A -85,B 0,C 180,E1 -22352.067,E2 -22352.067} C_VEL
LIN {X 0,Y 273.726,Z 580.258,A -85,B 0,C 180,E1 -22353.065,E2 -22353.065} C_VEL
LIN {X 0,Y 278.95,Z 565.755,A -85,B 0,C 180,E1 -22353.837,E2 -22353.837} C_VEL
LIN {X 0,Y 282.947,Z 551.791,A -85,B 0,C 180,E1 -22354.415,E2 -22354.415} C_VEL
LIN {X 0,Y 288.869,Z 524.63,A -85,B 0,C 180,E1 -22355.279,E2 -22355.279} C_VEL
LIN {X 0,Y 288.859,Z 524.71,A -85,B 0,C 180,E1 -22355.357,E2 -22355.357} C_VEL
LIN {X 0,Y 286.155,Z 537.436,A -85,B 0,C 180,E1 -22355.744,E2 -22355.744} C_VEL
LIN {X 0,Y 284.378,Z 545.685,A -85,B 0,C 180,E1 -22355.908,E2 -22355.908} C_VEL
LIN {X 0,Y 280.869,Z 559.248,A -85,B 0,C 180,E1 -22355.753,E2 -22355.753} C_VEL
LIN {X 0,Y 277.605,Z 569.335,A -85,B 0,C 180,E1 -22355.627,E2 -22355.627} C_VEL
LIN {X 0,Y 274.875,Z 576.802,A -85,B 0,C 180,E1 -22355.732,E2 -22355.732} C_VEL
LIN {X 0,Y 273.942,Z 579.172,A -85,B 0,C 180,E1 -22355.833,E2 -22355.833} C_VEL
LIN {X 0,Y 267.328,Z 594.34,A -85,B 0,C 180,E1 -22356.691,E2 -22356.691} C_VEL
LIN {X 0,Y 259.974,Z 608.452,A -85,B 0,C 180,E1 -22357.743,E2 -22357.743} C_VEL
LIN {X 0,Y 251.542,Z 622.581,A -85,B 0,C 180,E1 -22359.163,E2 -22359.163} C_VEL
LIN {X 0,Y 243.413,Z 634.451,A -85,B 0,C 180,E1 -22360.717,E2 -22360.717} C_VEL
LIN {X 0,Y 234.355,Z 646.393,A -85,B 0,C 180,E1 -22362.713,E2 -22362.713} C_VEL
LIN {X 0,Y 224.677,Z 657.885,A -85,B 0,C 180,E1 -22365.264,E2 -22365.264} C_VEL
LIN {X 0,Y 216.747,Z 666.395,A -85,B 0,C 180,E1 -22367.712,E2 -22367.712} C_VEL
LIN {X 0,Y 208.276,Z 674.866,A -85,B 0,C 180,E1 -22370.816,E2 -22370.816} C_VEL
LIN {X 0,Y 199.949,Z 682.511,A -85,B 0,C 180,E1 -22374.549,E2 -22374.549} C_VEL
LIN {X 0,Y 193.538,Z 688.081,A -85,B 0,C 180,E1 -22378.225,E2 -22378.225} C_VEL
LIN {X 0,Y 186.833,Z 693.474,A -85,B 0,C 180,E1 -22383.163,E2 -22383.163} C_VEL
LIN {X 0,Y 181.725,Z 697.041,A -85,B 0,C 180,E1 -22388.15,E2 -22388.15} C_VEL
LIN {X 0,Y 179.353,Z 698.658,A -85,B 0,C 180,E1 -22391.727,E2 -22391.727} C_VEL
LIN {X 0,Y 177.274,Z 699.623,A -85,B 0,C 180,E1 -22396.236,E2 -22396.236} C_VEL
LIN {X 0,Y 176.257,Z 699.557,A -85,B 0,C 180,E1 -22400.819,E2 -22400.819} C_VEL
LIN {X 0,Y 176.045,Z 698.417,A -85,B 0,C 180,E1 -22405.417,E2 -22405.417} C_VEL
LIN {X 0,Y 176.193,Z 697.406,A -85,B 0,C 180,E1 -22407.711,E2 -22407.711} C_VEL
LIN {X 0,Y 176.338,Z 696.047,A -85,B 0,C 180,E1 -22409.997,E2 -22409.997} C_VEL
LIN {X 0,Y 176.283,Z 693.311,A -85,B 0,C 180,E1 -22413.461,E2 -22413.461} C_VEL
LIN {X 0,Y 176.325,Z 689.833,A -85,B 0,C 180,E1 -22416.864,E2 -22416.864} C_VEL
LIN {X 0,Y 176.759,Z 683.766,A -85,B 0,C 180,E1 -22421.463,E2 -22421.463} C_VEL
LIN {X 0,Y 177.769,Z 677.05,A -85,B 0,C 180,E1 -22425.474,E2 -22425.474} C_VEL
LIN {X 0,Y 179.33,Z 669.164,A -85,B 0,C 180,E1 -22429.305,E2 -22429.305} C_VEL
LIN {X 0,Y 181.742,Z 658.884,A -85,B 0,C 180,E1 -22433.348,E2 -22433.348} C_VEL
LIN {X 0,Y 184.243,Z 648.663,A -85,B 0,C 180,E1 -22436.625,E2 -22436.625} C_VEL
LIN {X 0,Y 187.197,Z 636.955,A -85,B 0,C 180,E1 -22439.711,E2 -22439.711} C_VEL
LIN {X 0,Y 190.271,Z 624.558,A -85,B 0,C 180,E1 -22442.379,E2 -22442.379} C_VEL
LIN {X 0,Y 193.596,Z 610.213,A -85,B 0,C 180,E1 -22444.869,E2 -22444.869} C_VEL
LIN {X 0,Y 196.549,Z 596.27,A -85,B 0,C 180,E1 -22446.789,E2 -22446.789} C_VEL
LIN {X 0,Y 199.233,Z 581.092,A -85,B 0,C 180,E1 -22448.438,E2 -22448.438} C_VEL
LIN {X 0,Y 201.731,Z 564.47,A -85,B 0,C 180,E1 -22449.773,E2 -22449.773} C_VEL
LIN {X 0,Y 203.526,Z 547.052,A -85,B 0,C 180,E1 -22450.743,E2 -22450.743} C_VEL
LIN {X 0,Y 210.744,Z 465.226,A -85,B 0,C 180,E1 -22454.494,E2 -22454.494} C_VEL
LIN {X 0,Y 201.993,Z 442.576,A -85,B 0,C 180,E1 -22457.255,E2 -22457.255} C_VEL
LIN {X 0,Y 192.63,Z 420.837,A -85,B 0,C 180,E1 -22460.407,E2 -22460.407} C_VEL
LIN {X 0,Y 186.14,Z 407.049,A -85,B 0,C 180,E1 -22462.708,E2 -22462.708} C_VEL
LIN {X 0,Y 180.004,Z 396.503,A -85,B 0,C 180,E1 -22464.903,E2 -22464.903} C_VEL
LIN {X 0,Y 178.663,Z 393.865,A -85,B 0,C 180,E1 -22465.421,E2 -22465.421} C_VEL
LIN {X 0,Y 178.468,Z 392.882,A -85,B 0,C 180,E1 -22465.648,E2 -22465.648} C_VEL
LIN {X 0,Y 178.469,Z 392.878,A -85,B 0,C 180,E1 -22470.029,E2 -22470.029} C_VEL
LIN {X 0,Y 178.453,Z 392.871,A -85,B 0,C 180,E1 -22474.923,E2 -22474.923} C_VEL
LIN {X 0,Y 178.542,Z 392.854,A -85,B 0,C 180,E1 -22480.847,E2 -22480.847} C_VEL
LIN {X 0,Y 178.62,Z 392.858,A -85,B 0,C 180,E1 -22486.346,E2 -22486.346} C_VEL
LIN {X 0,Y 178.89,Z 392.811,A -85,B 0,C 180,E1 -22490.959,E2 -22490.959} C_VEL
LIN {X 0,Y 179.11,Z 392.793,A -85,B 0,C 180,E1 -22497.752,E2 -22497.752} C_VEL
LIN {X 0,Y 179.332,Z 392.774,A -85,B 0,C 180,E1 -22500.001,E2 -22500.001} C_VEL
LIN {X 0,Y 178.82,Z 392.832,A -85,B 0,C 180,E1 -22504.509,E2 -22504.509} C_VEL
LIN {X 0,Y 178.893,Z 392.821,A -85,B 0,C 180,E1 -22509.042,E2 -22509.042} C_VEL
LIN {X 0,Y 178.621,Z 392.86,A -85,B 0,C 180,E1 -22513.656,E2 -22513.656} C_VEL
LIN {X 0,Y 178.544,Z 392.864,A -85,B 0,C 180,E1 -22519.154,E2 -22519.154} C_VEL
LIN {X 0,Y 178.455,Z 392.871,A -85,B 0,C 180,E1 -22525.078,E2 -22525.078} C_VEL
LIN {X 0,Y 178.45,Z 392.879,A -85,B 0,C 180,E1 -22530.797,E2 -22530.797} C_VEL
LIN {X 0,Y 178.473,Z 392.866,A -85,B 0,C 180,E1 -22534.221,E2 -22534.221} C_VEL
LIN {X 0,Y 178.379,Z 392.888,A -85,B 0,C 180,E1 -22539.08,E2 -22539.08} C_VEL
LIN {X 0,Y 178.386,Z 392.877,A -85,B 0,C 180,E1 -22542.05,E2 -22542.05} C_VEL
LIN {X 0,Y 178.384,Z 392.886,A -85,B 0,C 180,E1 -22545.168,E2 -22545.168} C_VEL
LIN {X 0,Y 178.39,Z 392.885,A -85,B 0,C 180,E1 -22548.465,E2 -22548.465} C_VEL
LIN {X 0,Y 178.413,Z 392.885,A -85,B 0,C 180,E1 -22553.786,E2 -22553.786} C_VEL
LIN {X 0,Y 178.479,Z 392.874,A -85,B 0,C 180,E1 -22556.55,E2 -22556.55} C_VEL
LIN {X 0,Y 178.437,Z 392.884,A -85,B 0,C 180,E1 -22561.799,E2 -22561.799} C_VEL
LIN {X 0,Y 178.502,Z 392.869,A -85,B 0,C 180,E1 -22564.9,E2 -22564.9} C_VEL
LIN {X 0,Y 178.562,Z 392.865,A -85,B 0,C 180,E1 -22570.844,E2 -22570.844} C_VEL
LIN {X 0,Y 178.647,Z 392.833,A -85,B 0,C 180,E1 -22576.351,E2 -22576.351} C_VEL
LIN {X 0,Y 178.906,Z 392.824,A -85,B 0,C 180,E1 -22580.963,E2 -22580.963} C_VEL
LIN {X 0,Y 179.127,Z 392.795,A -85,B 0,C 180,E1 -22587.755,E2 -22587.755} C_VEL
LIN {X 0,Y 179.348,Z 392.77,A -85,B 0,C 180,E1 -22590.003,E2 -22590.003} C_VEL
LIN {X 0,Y 178.84,Z 392.83,A -85,B 0,C 180,E1 -22594.511,E2 -22594.511} C_VEL
LIN {X 0,Y 178.91,Z 392.815,A -85,B 0,C 180,E1 -22599.044,E2 -22599.044} C_VEL
LIN {X 0,Y 178.634,Z 392.851,A -85,B 0,C 180,E1 -22603.657,E2 -22603.657} C_VEL
LIN {X 0,Y 178.595,Z 392.865,A -85,B 0,C 180,E1 -22606.286,E2 -22606.286} C_VEL
LIN {X 0,Y 179.603,Z 395.696,A -85,B 0,C 180,E1 -22606.777,E2 -22606.777} C_VEL
LIN {X 0,Y 181.086,Z 397.944,A -85,B 0,C 180,E1 -22607.289,E2 -22607.289} C_VEL
LIN {X 0,Y 190.397,Z 414.76,A -85,B 0,C 180,E1 -22610.547,E2 -22610.547} C_VEL
LIN {X 0,Y 199.03,Z 431.422,A -85,B 0,C 180,E1 -22613.301,E2 -22613.301} C_VEL
LIN {X 0,Y 208.424,Z 451.101,A -85,B 0,C 180,E1 -22616.116,E2 -22616.116} C_VEL
LIN {X 0,Y 210.718,Z 457.319,A -85,B 0,C 180,E1 -22616.834,E2 -22616.834} C_VEL
LIN {X 0,Y 202.688,Z 546.047,A -85,B 0,C 180,E1 -22620.91,E2 -22620.91} C_VEL
LIN {X 0,Y 200.682,Z 562.151,A -85,B 0,C 180,E1 -22622.026,E2 -22622.026} C_VEL
LIN {X 0,Y 198.203,Z 578.214,A -85,B 0,C 180,E1 -22623.562,E2 -22623.562} C_VEL
LIN {X 0,Y 195.126,Z 594.289,A -85,B 0,C 180,E1 -22625.571,E2 -22625.571} C_VEL
LIN {X 0,Y 191.989,Z 608.829,A -85,B 0,C 180,E1 -22627.891,E2 -22627.891} C_VEL
LIN {X 0,Y 188.723,Z 622.648,A -85,B 0,C 180,E1 -22630.644,E2 -22630.644} C_VEL
LIN {X 0,Y 185.816,Z 634.234,A -85,B 0,C 180,E1 -22633.485,E2 -22633.485} C_VEL
LIN {X 0,Y 182.911,Z 645.675,A -85,B 0,C 180,E1 -22636.894,E2 -22636.894} C_VEL
LIN {X 0,Y 180.76,Z 654.866,A -85,B 0,C 180,E1 -22640.238,E2 -22640.238} C_VEL
LIN {X 0,Y 178.866,Z 663.188,A -85,B 0,C 180,E1 -22643.886,E2 -22643.886} C_VEL
LIN {X 0,Y 177.317,Z 671.433,A -85,B 0,C 180,E1 -22648.32,E2 -22648.32} C_VEL
LIN {X 0,Y 176.573,Z 676.258,A -85,B 0,C 180,E1 -22651.469,E2 -22651.469} C_VEL
LIN {X 0,Y 175.936,Z 680.933,A -85,B 0,C 180,E1 -22655.2,E2 -22655.2} C_VEL
LIN {X 0,Y 175.574,Z 684.622,A -85,B 0,C 180,E1 -22658.883,E2 -22658.883} C_VEL
LIN {X 0,Y 175.65,Z 688.205,A -85,B 0,C 180,E1 -22663.806,E2 -22663.806} C_VEL
LIN {X 0,Y 176.311,Z 690.357,A -85,B 0,C 180,E1 -22668.503,E2 -22668.503} C_VEL
LIN {X 0,Y 177.825,Z 691.288,A -85,B 0,C 180,E1 -22673.19,E2 -22673.19} C_VEL
LIN {X 0,Y 180.122,Z 691.068,A -85,B 0,C 180,E1 -22677.763,E2 -22677.763} C_VEL
LIN {X 0,Y 183.452,Z 689.751,A -85,B 0,C 180,E1 -22682.195,E2 -22682.195} C_VEL
LIN {X 0,Y 187.838,Z 687.363,A -85,B 0,C 180,E1 -22686.444,E2 -22686.444} C_VEL
LIN {X 0,Y 193.164,Z 683.801,A -85,B 0,C 180,E1 -22690.481,E2 -22690.481} C_VEL
LIN {X 0,Y 199.488,Z 679.071,A -85,B 0,C 180,E1 -22694.276,E2 -22694.276} C_VEL
LIN {X 0,Y 206.81,Z 673.029,A -85,B 0,C 180,E1 -22697.809,E2 -22697.809} C_VEL
LIN {X 0,Y 214.918,Z 665.63,A -85,B 0,C 180,E1 -22701.082,E2 -22701.082} C_VEL
LIN {X 0,Y 223.915,Z 656.61,A -85,B 0,C 180,E1 -22704.081,E2 -22704.081} C_VEL
LIN {X 0,Y 232.405,Z 647.111,A -85,B 0,C 180,E1 -22706.49,E2 -22706.49} C_VEL
LIN {X 0,Y 240.755,Z 636.842,A -85,B 0,C 180,E1 -22708.57,E2 -22708.57} C_VEL
LIN {X 0,Y 250.15,Z 623.753,A -85,B 0,C 180,E1 -22710.612,E2 -22710.612} C_VEL
LIN {X 0,Y 258.289,Z 610.836,A -85,B 0,C 180,E1 -22712.16,E2 -22712.16} C_VEL
